Yaskawa INFORM job: DEMO_ROOF_SIDE_0625_3PAINT_60.JBI

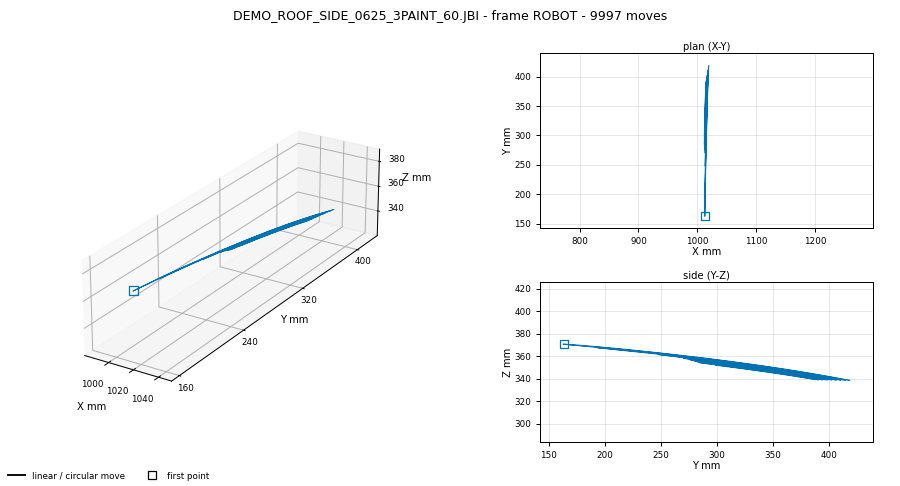
[picture p0: tool path of DEMO_ROOF_SIDE_0625_3PAINT_60.JBI in frame ROBOT, 9997 of 9997 moves have a stored position in this frame; points joined in program order, loops and branches not executed]
/JOB
//NAME DEMO_ROOF_SIDE_0625_3PAINT60
//POS
///NPOS 9997,0,0,0,0,0
///TOOL 0
///USER 0
///POSTYPE ROBOT
///RECTAN
///RCONF 1,0,0,0,0,0,0,0,0,0,0,0,0,0,0,0,0,0,0,0,0,0,0,0
C00000=1012.769,163.450,371.044,166.546,56.934,160.427
C00001=1012.773,163.699,371.026,166.549,56.922,160.426
C00002=1012.776,163.949,371.006,166.553,56.910,160.424
C00003=1012.781,164.198,370.986,166.556,56.898,160.423
C00004=1012.783,164.447,370.967,166.560,56.886,160.421
C00005=1012.788,164.696,370.948,166.563,56.875,160.420
C00006=1012.791,164.945,370.928,166.568,56.863,160.418
C00007=1012.795,165.195,370.908,166.571,56.851,160.417
C00008=1012.798,165.444,370.889,166.574,56.839,160.415
C00009=1012.802,165.693,370.869,166.578,56.827,160.414
C00010=1012.806,165.942,370.850,166.581,56.815,160.412
C00011=1012.810,166.191,370.830,166.586,56.803,160.411
C00012=1012.813,166.441,370.811,166.589,56.791,160.409
C00013=1012.817,166.690,370.791,166.592,56.779,160.408
C00014=1012.820,166.939,370.771,166.596,56.767,160.406
C00015=1012.825,167.188,370.752,166.599,56.756,160.405
C00016=1012.828,167.437,370.733,166.604,56.743,160.403
C00017=1012.832,167.686,370.713,166.607,56.732,160.402
C00018=1012.836,167.936,370.693,166.610,56.720,160.400
C00019=1012.839,168.185,370.673,166.614,56.707,160.398
C00020=1012.843,168.434,370.654,166.617,56.695,160.397
C00021=1012.846,168.684,370.635,166.621,56.683,160.395
C00022=1012.851,168.933,370.615,166.624,56.671,160.394
C00023=1012.854,169.182,370.595,166.629,56.659,160.393
C00024=1012.858,169.431,370.575,166.632,56.647,160.391
C00025=1012.862,169.680,370.556,166.636,56.635,160.390
C00026=1012.866,169.930,370.536,166.639,56.623,160.388
C00027=1012.870,170.208,370.514,166.644,56.609,160.386
C00028=1012.874,170.487,370.492,166.648,56.596,160.385
C00029=1012.878,170.766,370.470,166.652,56.583,160.383
C00030=1012.882,171.045,370.448,166.656,56.569,160.381
C00031=1012.887,171.294,370.428,166.661,56.557,160.380
C00032=1012.890,171.543,370.408,166.664,56.545,160.378
C00033=1012.894,171.793,370.389,166.668,56.532,160.377
C00034=1012.898,172.042,370.369,166.671,56.521,160.375
C00035=1012.902,172.292,370.349,166.675,56.509,160.374
C00036=1012.906,172.541,370.330,166.678,56.497,160.372
C00037=1012.910,172.790,370.310,166.683,56.485,160.371
C00038=1012.913,173.040,370.290,166.687,56.472,160.369
C00039=1012.917,173.288,370.271,166.690,56.460,160.367
C00040=1012.921,173.537,370.251,166.694,56.448,160.366
C00041=1012.925,173.786,370.231,166.699,56.436,160.365
C00042=1012.928,174.036,370.211,166.701,56.424,160.363
C00043=1012.932,174.285,370.191,166.706,56.411,160.361
C00044=1012.936,174.534,370.172,166.710,56.399,160.360
C00045=1012.940,174.783,370.151,166.713,56.388,160.358
C00046=1012.944,175.032,370.132,166.717,56.375,160.357
C00047=1012.948,175.282,370.112,166.721,56.363,160.355
C00048=1012.952,175.531,370.092,166.725,56.351,160.354
C00049=1012.956,175.780,370.072,166.729,56.339,160.352
C00050=1012.960,176.030,370.052,166.733,56.326,160.351
C00051=1012.964,176.279,370.033,166.737,56.314,160.349
C00052=1012.968,176.527,370.012,166.741,56.302,160.348
C00053=1012.972,176.776,369.993,166.744,56.289,160.346
C00054=1012.976,177.026,369.973,166.749,56.277,160.345
C00055=1012.979,177.275,369.952,166.753,56.265,160.343
C00056=1012.984,177.524,369.933,166.757,56.252,160.342
C00057=1012.987,177.773,369.913,166.760,56.241,160.340
C00058=1012.992,178.022,369.893,166.765,56.229,160.339
C00059=1012.995,178.272,369.873,166.769,56.216,160.337
C00060=1012.999,178.521,369.853,166.773,56.204,160.336
C00061=1013.004,178.770,369.833,166.777,56.191,160.334
C00062=1013.007,179.019,369.813,166.780,56.179,160.332
C00063=1013.012,179.268,369.794,166.785,56.167,160.331
C00064=1013.015,179.517,369.774,166.788,56.155,160.329
C00065=1013.019,179.767,369.753,166.793,56.142,160.328
C00066=1013.023,180.016,369.734,166.797,56.130,160.326
C00067=1013.028,180.265,369.713,166.801,56.118,160.325
C00068=1013.032,180.514,369.693,166.805,56.105,160.323
C00069=1013.036,180.764,369.673,166.809,56.093,160.322
C00070=1013.039,181.013,369.653,166.813,56.081,160.320
C00071=1013.044,181.261,369.633,166.817,56.068,160.319
C00072=1013.047,181.511,369.613,166.821,56.056,160.317
C00073=1013.050,181.760,369.592,166.826,56.044,160.316
C00074=1013.055,182.010,369.571,166.830,56.032,160.314
C00075=1013.059,182.259,369.550,166.833,56.020,160.313
C00076=1013.062,182.508,369.530,166.837,56.008,160.311
C00077=1013.066,182.757,369.509,166.842,55.996,160.310
C00078=1013.069,183.006,369.489,166.846,55.984,160.309
C00079=1013.073,183.255,369.468,166.849,55.972,160.307
C00080=1013.076,183.504,369.447,166.854,55.960,160.306
C00081=1013.080,183.753,369.427,166.858,55.947,160.304
C00082=1013.084,184.003,369.406,166.863,55.935,160.303
C00083=1013.088,184.252,369.385,166.866,55.924,160.301
C00084=1013.091,184.501,369.363,166.870,55.911,160.300
C00085=1013.095,184.750,369.343,166.874,55.899,160.298
C00086=1013.099,184.999,369.323,166.879,55.887,160.297
C00087=1013.103,185.247,369.302,166.883,55.874,160.295
C00088=1013.106,185.497,369.281,166.887,55.862,160.294
C00089=1013.110,185.747,369.260,166.891,55.851,160.292
C00090=1013.114,185.995,369.239,166.895,55.839,160.291
C00091=1013.118,186.274,369.216,166.900,55.825,160.289
C00092=1013.122,186.553,369.192,166.904,55.811,160.287
C00093=1013.127,186.832,369.169,166.910,55.798,160.286
C00094=1013.131,187.111,369.146,166.915,55.784,160.284
C00095=1013.134,187.360,369.125,166.918,55.772,160.283
C00096=1013.139,187.610,369.104,166.922,55.759,160.281
C00097=1013.142,187.858,369.083,166.927,55.748,160.280
C00098=1013.146,188.107,369.063,166.931,55.736,160.278
C00099=1013.150,188.356,369.041,166.935,55.723,160.277
C00100=1013.154,188.606,369.020,166.940,55.711,160.275
C00101=1013.158,188.854,368.999,166.944,55.699,160.274
C00102=1013.162,189.103,368.979,166.948,55.686,160.272
C00103=1013.165,189.353,368.958,166.953,55.674,160.271
C00104=1013.169,189.602,368.937,166.957,55.662,160.270
C00105=1013.173,189.851,368.916,166.961,55.650,160.268
C00106=1013.176,190.100,368.895,166.966,55.638,160.267
C00107=1013.181,190.349,368.874,166.970,55.625,160.265
C00108=1013.185,190.598,368.853,166.975,55.613,160.264
C00109=1013.189,190.847,368.832,166.979,55.601,160.262
C00110=1013.192,191.097,368.810,166.983,55.588,160.261
C00111=1013.196,191.345,368.789,166.988,55.576,160.259
C00112=1013.200,191.594,368.769,166.992,55.564,160.258
C00113=1013.205,191.843,368.747,166.996,55.552,160.256
C00114=1013.208,192.092,368.726,167.001,55.540,160.255
C00115=1013.212,192.341,368.705,167.005,55.527,160.253
C00116=1013.216,192.591,368.684,167.010,55.515,160.252
C00117=1013.220,192.840,368.663,167.015,55.502,160.251
C00118=1013.224,193.088,368.642,167.019,55.490,160.249
C00119=1013.228,193.338,368.621,167.023,55.478,160.248
C00120=1013.232,193.587,368.600,167.028,55.466,160.246
C00121=1013.236,193.836,368.578,167.033,55.454,160.245
C00122=1013.240,194.085,368.558,167.037,55.441,160.243
C00123=1013.244,194.334,368.537,167.041,55.429,160.242
C00124=1013.248,194.583,368.516,167.045,55.417,160.240
C00125=1013.251,194.832,368.494,167.051,55.404,160.239
C00126=1013.256,195.082,368.473,167.055,55.392,160.237
C00127=1013.260,195.330,368.452,167.060,55.380,160.236
C00128=1013.263,195.580,368.431,167.064,55.367,160.234
C00129=1013.267,195.829,368.410,167.068,55.355,160.233
C00130=1013.271,196.078,368.389,167.073,55.343,160.231
C00131=1013.276,196.326,368.367,167.078,55.331,160.230
C00132=1013.279,196.576,368.346,167.082,55.318,160.229
C00133=1013.284,196.825,368.325,167.087,55.306,160.227
C00134=1013.288,197.074,368.304,167.091,55.293,160.226
C00135=1013.292,197.323,368.283,167.097,55.281,160.224
C00136=1013.295,197.572,368.261,167.101,55.269,160.223
C00137=1013.300,197.821,368.239,167.106,55.257,160.221
C00138=1013.304,198.070,368.219,167.110,55.244,160.220
C00139=1013.308,198.319,368.197,167.115,55.232,160.219
C00140=1013.312,198.568,368.176,167.120,55.219,160.217
C00141=1013.316,198.818,368.155,167.124,55.207,160.216
C00142=1013.320,199.067,368.133,167.128,55.195,160.214
C00143=1013.324,199.316,368.111,167.134,55.183,160.213
C00144=1013.328,199.565,368.089,167.138,55.170,160.211
C00145=1013.332,199.814,368.068,167.143,55.158,160.210
C00146=1013.336,200.063,368.045,167.148,55.146,160.209
C00147=1013.340,200.312,368.025,167.152,55.134,160.207
C00148=1013.344,200.561,368.002,167.157,55.122,160.206
C00149=1013.347,200.810,367.981,167.162,55.109,160.204
C00150=1013.352,201.059,367.959,167.166,55.097,160.203
C00151=1013.356,201.308,367.937,167.171,55.085,160.201
C00152=1013.359,201.557,367.915,167.176,55.072,160.200
C00153=1013.364,201.806,367.894,167.181,55.061,160.199
C00154=1013.367,202.055,367.872,167.185,55.048,160.197
C00155=1013.384,203.102,367.780,167.720,55.151,160.345
C00156=1013.390,203.386,367.754,167.725,55.138,160.343
C00157=1013.395,203.671,367.727,167.730,55.125,160.342
C00158=1013.402,203.957,367.700,167.736,55.113,160.340
C00159=1013.408,204.241,367.672,167.741,55.100,160.339
C00160=1013.412,204.490,367.649,167.746,55.089,160.337
C00161=1013.417,204.739,367.626,167.751,55.077,160.336
C00162=1013.422,204.988,367.602,167.755,55.066,160.335
C00163=1013.428,205.237,367.579,167.760,55.055,160.333
C00164=1013.433,205.486,367.555,167.764,55.045,160.332
C00165=1013.438,205.734,367.531,167.769,55.034,160.331
C00166=1013.443,205.983,367.508,167.773,55.022,160.329
C00167=1013.448,206.232,367.484,167.778,55.011,160.328
C00168=1013.453,206.481,367.460,167.782,55.001,160.327
C00169=1013.458,206.730,367.436,167.787,54.989,160.326
C00170=1013.463,206.978,367.412,167.791,54.979,160.324
C00171=1013.468,207.227,367.389,167.796,54.968,160.323
C00172=1013.473,207.476,367.365,167.800,54.957,160.322
C00173=1013.478,207.725,367.341,167.806,54.946,160.320
C00174=1013.483,207.973,367.317,167.810,54.935,160.319
C00175=1013.488,208.223,367.293,167.815,54.924,160.318
C00176=1013.493,208.451,367.271,167.818,54.914,160.316
C00177=1013.498,208.678,367.250,167.822,54.904,160.315
C00178=1013.502,208.907,367.228,167.827,54.894,160.314
C00179=1013.507,209.134,367.206,167.831,54.885,160.313
C00180=1013.511,209.362,367.184,167.835,54.875,160.312
C00181=1013.516,209.590,367.161,167.840,54.865,160.311
C00182=1013.520,209.818,367.139,167.844,54.855,160.310
C00183=1013.525,210.046,367.118,167.848,54.845,160.309
C00184=1013.530,210.294,367.093,167.852,54.835,160.307
C00185=1013.535,210.544,367.069,167.856,54.824,160.306
C00186=1013.540,210.792,367.045,167.862,54.813,160.305
C00187=1013.545,211.041,367.021,167.866,54.802,160.303
C00188=1013.550,211.290,366.997,167.871,54.791,160.302
C00189=1013.555,211.539,366.972,167.875,54.781,160.301
C00190=1013.560,211.788,366.948,167.880,54.771,160.300
C00191=1013.565,212.036,366.924,167.885,54.760,160.299
C00192=1013.570,212.285,366.900,167.889,54.749,160.297
C00193=1013.576,212.534,366.876,167.893,54.739,160.296
C00194=1013.580,212.783,366.851,167.898,54.728,160.295
C00195=1013.586,213.032,366.827,167.903,54.718,160.294
C00196=1013.591,213.280,366.803,167.907,54.707,160.292
C00197=1013.596,213.529,366.779,167.911,54.697,160.291
C00198=1013.601,213.778,366.755,167.917,54.686,160.290
C00199=1013.606,214.027,366.730,167.921,54.676,160.289
C00200=1013.611,214.275,366.706,167.925,54.665,160.287
C00201=1013.616,214.524,366.681,167.931,54.654,160.286
C00202=1013.622,214.773,366.657,167.935,54.644,160.285
C00203=1013.626,215.021,366.632,167.939,54.634,160.284
C00204=1013.631,215.271,366.609,167.944,54.623,160.282
C00205=1013.636,215.519,366.585,167.949,54.613,160.281
C00206=1013.642,215.769,366.560,167.954,54.602,160.280
C00207=1013.648,216.017,366.536,167.958,54.592,160.279
C00208=1013.652,216.266,366.511,167.963,54.581,160.278
C00209=1013.657,216.515,366.487,167.968,54.571,160.277
C00210=1013.663,216.763,366.462,167.972,54.561,160.275
C00211=1013.668,217.012,366.438,167.977,54.550,160.274
C00212=1013.673,217.261,366.413,167.982,54.539,160.273
C00213=1013.678,217.509,366.389,167.987,54.529,160.272
C00214=1013.683,217.758,366.365,167.991,54.519,160.271
C00215=1013.688,218.007,366.340,167.995,54.509,160.269
C00216=1013.694,218.258,366.315,168.000,54.498,160.268
C00217=1013.699,218.511,366.289,168.005,54.488,160.267
C00218=1013.704,218.764,366.264,168.010,54.478,160.266
C00219=1013.709,219.015,366.239,168.014,54.468,160.265
C00220=1013.714,219.263,366.215,168.019,54.457,160.263
C00221=1013.719,219.513,366.189,168.023,54.447,160.262
C00222=1013.724,219.762,366.165,168.028,54.437,160.261
C00223=1013.729,220.010,366.140,168.033,54.427,160.260
C00224=1013.735,220.259,366.115,168.038,54.417,160.259
C00225=1013.739,220.507,366.090,168.043,54.407,160.258
C00226=1013.745,220.757,366.066,168.047,54.396,160.257
C00227=1013.750,221.005,366.040,168.052,54.386,160.256
C00228=1013.755,221.254,366.016,168.056,54.377,160.254
C00229=1013.760,221.503,365.991,168.061,54.367,160.253
C00230=1013.765,221.750,365.966,168.065,54.356,160.252
C00231=1013.770,222.000,365.941,168.070,54.346,160.251
C00232=1013.776,222.249,365.917,168.075,54.337,160.250
C00233=1013.781,222.497,365.891,168.080,54.327,160.249
C00234=1013.786,222.746,365.867,168.084,54.316,160.247
C00235=1013.791,222.995,365.842,168.090,54.306,160.247
C00236=1013.797,223.243,365.817,168.094,54.296,160.245
C00237=1013.801,223.492,365.792,168.099,54.286,160.244
C00238=1013.807,223.741,365.767,168.104,54.277,160.243
C00239=1013.812,223.990,365.742,168.108,54.266,160.242
C00240=1013.817,224.238,365.717,168.113,54.256,160.241
C00241=1013.823,224.487,365.692,168.118,54.246,160.240
C00242=1013.827,224.736,365.667,168.122,54.237,160.239
C00243=1013.833,224.984,365.642,168.127,54.227,160.238
C00244=1013.838,225.234,365.616,168.132,54.217,160.237
C00245=1013.844,225.482,365.592,168.137,54.207,160.236
C00246=1013.848,225.730,365.567,168.141,54.197,160.234
C00247=1013.854,225.979,365.541,168.146,54.187,160.233
C00248=1013.859,226.228,365.516,168.151,54.177,160.232
C00249=1013.864,226.476,365.491,168.156,54.168,160.231
C00250=1013.869,226.725,365.465,168.161,54.158,160.230
C00251=1013.875,226.974,365.441,168.165,54.148,160.229
C00252=1013.880,227.223,365.415,168.170,54.139,160.228
C00253=1013.885,227.471,365.389,168.174,54.129,160.227
C00254=1013.890,227.720,365.364,168.179,54.119,160.226
C00255=1013.895,227.969,365.338,168.184,54.110,160.225
C00256=1013.901,228.217,365.313,168.188,54.100,160.224
C00257=1013.906,228.466,365.288,168.193,54.090,160.222
C00258=1013.911,228.715,365.263,168.198,54.080,160.221
C00259=1013.916,228.963,365.237,168.203,54.071,160.221
C00260=1013.922,229.212,365.212,168.208,54.061,160.219
C00261=1013.927,229.460,365.186,168.213,54.052,160.218
C00262=1013.932,229.709,365.160,168.217,54.042,160.217
C00263=1013.937,229.957,365.135,168.222,54.033,160.216
C00264=1013.942,230.206,365.110,168.227,54.023,160.215
C00265=1013.947,230.455,365.084,168.231,54.014,160.214
C00266=1013.952,230.704,365.058,168.236,54.004,160.213
C00267=1013.957,230.952,365.032,168.242,53.995,160.212
C00268=1013.962,231.201,365.007,168.245,53.985,160.211
C00269=1013.968,231.450,364.981,168.250,53.976,160.210
C00270=1013.973,231.698,364.955,168.256,53.967,160.209
C00271=1013.978,231.947,364.929,168.260,53.957,160.208
C00272=1013.983,232.195,364.904,168.265,53.947,160.207
C00273=1013.989,232.444,364.879,168.269,53.938,160.206
C00274=1013.994,232.692,364.853,168.274,53.929,160.205
C00275=1013.999,232.941,364.827,168.280,53.920,160.204
C00276=1014.005,233.188,364.802,168.284,53.910,160.203
C00277=1014.010,233.433,364.776,168.289,53.901,160.202
C00278=1014.014,233.680,364.750,168.294,53.892,160.201
C00279=1014.020,233.927,364.725,168.299,53.882,160.200
C00280=1014.025,234.173,364.699,168.303,53.873,160.199
C00281=1014.030,234.419,364.674,168.308,53.864,160.198
C00282=1014.036,234.665,364.648,168.313,53.854,160.197
C00283=1014.041,234.911,364.622,168.317,53.846,160.196
C00284=1014.046,235.159,364.597,168.322,53.836,160.195
C00285=1014.051,235.408,364.571,168.327,53.827,160.194
C00286=1014.057,235.657,364.544,168.333,53.818,160.193
C00287=1014.062,235.905,364.519,168.336,53.809,160.192
C00288=1014.067,236.154,364.493,168.342,53.800,160.191
C00289=1014.073,236.403,364.467,168.347,53.790,160.190
C00290=1014.078,236.651,364.441,168.351,53.781,160.189
C00291=1014.083,236.900,364.415,168.356,53.772,160.189
C00292=1014.089,237.149,364.389,168.361,53.762,160.187
C00293=1014.094,237.397,364.363,168.365,53.754,160.186
C00294=1014.099,237.646,364.337,168.370,53.744,160.185
C00295=1014.105,237.894,364.311,168.376,53.735,160.185
C00296=1014.110,238.143,364.285,168.381,53.726,160.184
C00297=1014.115,238.392,364.259,168.385,53.717,160.183
C00298=1014.121,238.639,364.233,168.390,53.708,160.182
C00299=1014.126,238.888,364.207,168.395,53.699,160.181
C00300=1014.131,239.137,364.180,168.400,53.690,160.180
C00301=1014.136,239.386,364.154,168.405,53.681,160.179
C00302=1014.142,239.633,364.127,168.410,53.673,160.178
C00303=1014.146,239.883,364.101,168.414,53.663,160.177
C00304=1014.152,240.131,364.074,168.419,53.654,160.176
C00305=1014.157,240.379,364.049,168.424,53.645,160.175
C00306=1014.163,240.628,364.022,168.430,53.636,160.174
C00307=1014.168,240.877,363.995,168.434,53.628,160.173
C00308=1014.173,241.125,363.969,168.439,53.619,160.173
C00309=1014.178,241.374,363.943,168.444,53.610,160.172
C00310=1014.183,241.622,363.916,168.449,53.601,160.171
C00311=1014.189,241.871,363.889,168.453,53.592,160.170
C00312=1014.194,242.120,363.863,168.459,53.583,160.169
C00313=1014.200,242.367,363.837,168.464,53.574,160.168
C00314=1014.205,242.616,363.810,168.468,53.566,160.167
C00315=1014.210,242.865,363.784,168.474,53.557,160.166
C00316=1014.215,243.114,363.757,168.478,53.548,160.165
C00317=1014.221,243.362,363.730,168.482,53.540,160.164
C00318=1014.225,243.610,363.703,168.488,53.531,160.164
C00319=1014.231,243.858,363.677,168.493,53.523,160.163
C00320=1014.236,244.107,363.649,168.498,53.514,160.162
C00321=1014.241,244.356,363.623,168.502,53.505,160.161
C00322=1014.247,244.605,363.596,168.508,53.496,160.160
C00323=1014.252,244.853,363.569,168.512,53.488,160.159
C00324=1014.257,245.101,363.543,168.518,53.479,160.159
C00325=1014.262,245.350,363.515,168.522,53.471,160.158
C00326=1014.267,245.598,363.488,168.527,53.462,160.157
C00327=1014.273,245.847,363.461,168.532,53.453,160.156
C00328=1014.278,246.095,363.434,168.537,53.445,160.155
C00329=1014.284,246.344,363.408,168.542,53.436,160.154
C00330=1014.289,246.592,363.380,168.547,53.428,160.153
C00331=1014.294,246.841,363.353,168.553,53.420,160.153
C00332=1014.299,247.089,363.326,168.557,53.411,160.152
C00333=1014.304,247.337,363.300,168.561,53.403,160.151
C00334=1014.310,247.586,363.273,168.567,53.394,160.150
C00335=1014.315,247.834,363.246,168.572,53.386,160.149
C00336=1014.320,248.077,363.220,168.577,53.378,160.149
C00337=1014.325,248.321,363.193,168.582,53.369,160.148
C00338=1014.331,248.563,363.167,168.587,53.361,160.147
C00339=1014.336,248.806,363.140,168.591,53.352,160.146
C00340=1014.341,249.049,363.115,168.596,53.345,160.145
C00341=1014.346,249.291,363.087,168.600,53.336,160.144
C00342=1014.352,249.534,363.061,168.606,53.328,160.144
C00343=1014.356,249.777,363.035,168.611,53.320,160.143
C00344=1014.362,250.025,363.008,168.616,53.311,160.142
C00345=1014.367,250.274,362.981,168.621,53.303,160.142
C00346=1014.373,250.522,362.953,168.626,53.295,160.141
C00347=1014.378,250.770,362.926,168.631,53.287,160.140
C00348=1014.383,251.019,362.899,168.636,53.278,160.139
C00349=1014.389,251.267,362.872,168.641,53.270,160.138
C00350=1014.394,251.516,362.845,168.645,53.261,160.137
C00351=1014.400,251.765,362.817,168.651,53.253,160.137
C00352=1014.406,252.013,362.790,168.656,53.245,160.136
C00353=1014.411,252.262,362.763,168.662,53.236,160.135
C00354=1014.417,252.510,362.736,168.667,53.229,160.134
C00355=1014.422,252.759,362.709,168.671,53.220,160.134
C00356=1014.427,253.007,362.681,168.677,53.212,160.133
C00357=1014.433,253.255,362.654,168.681,53.203,160.132
C00358=1014.438,253.504,362.627,168.686,53.195,160.131
C00359=1014.444,253.752,362.600,168.692,53.187,160.131
C00360=1014.450,254.001,362.572,168.696,53.179,160.130
C00361=1014.455,254.250,362.545,168.701,53.171,160.129
C00362=1014.461,254.497,362.517,168.707,53.163,160.128
C00363=1014.466,254.746,362.490,168.712,53.155,160.128
C00364=1014.472,254.994,362.464,168.717,53.146,160.127
C00365=1014.477,255.243,362.436,168.722,53.138,160.126
C00366=1014.483,255.492,362.408,168.727,53.130,160.125
C00367=1014.489,255.740,362.381,168.732,53.122,160.124
C00368=1014.494,255.988,362.353,168.738,53.114,160.124
C00369=1014.499,256.237,362.327,168.743,53.106,160.123
C00370=1014.505,256.485,362.298,168.747,53.098,160.122
C00371=1014.510,256.734,362.271,168.753,53.090,160.122
C00372=1014.516,256.982,362.244,168.758,53.081,160.121
C00373=1014.522,257.231,362.217,168.763,53.073,160.120
C00374=1014.527,257.479,362.188,168.768,53.066,160.119
C00375=1014.533,257.728,362.162,168.773,53.057,160.119
C00376=1014.539,257.976,362.134,168.778,53.050,160.118
C00377=1014.545,258.225,362.107,168.783,53.042,160.117
C00378=1014.550,258.473,362.079,168.789,53.034,160.117
C00379=1014.555,258.721,362.051,168.794,53.026,160.116
C00380=1014.561,258.969,362.024,168.799,53.017,160.115
C00381=1014.567,259.218,361.996,168.803,53.009,160.114
C00382=1014.573,259.466,361.968,168.809,53.001,160.114
C00383=1014.578,259.714,361.941,168.814,52.993,160.113
C00384=1014.584,259.962,361.913,168.820,52.986,160.112
C00385=1014.590,260.211,361.885,168.825,52.979,160.112
C00386=1014.595,260.459,361.857,168.829,52.971,160.111
C00387=1014.600,260.707,361.829,168.835,52.963,160.110
C00388=1014.606,260.956,361.801,168.840,52.955,160.110
C00389=1014.611,261.205,361.773,168.845,52.947,160.109
C00390=1014.617,261.453,361.745,168.851,52.940,160.108
C00391=1014.623,261.701,361.717,168.856,52.932,160.108
C00392=1014.627,261.950,361.689,168.860,52.924,160.107
C00393=1014.633,262.198,361.661,168.865,52.916,160.106
C00394=1014.639,262.447,361.632,168.872,52.909,160.106
C00395=1014.644,262.695,361.604,168.877,52.901,160.105
C00396=1014.650,262.936,361.577,168.882,52.893,160.104
C00397=1014.655,263.178,361.550,168.887,52.886,160.104
C00398=1014.660,263.420,361.522,168.892,52.879,160.103
C00399=1014.666,263.662,361.495,168.896,52.872,160.102
C00400=1014.671,263.903,361.467,168.901,52.864,160.102
C00401=1014.677,264.146,361.440,168.907,52.857,160.101
C00402=1014.682,264.387,361.413,168.912,52.849,160.100
C00403=1014.687,264.629,361.385,168.917,52.842,160.100
C00404=1014.693,264.877,361.356,168.922,52.834,160.099
C00405=1014.699,265.125,361.328,168.927,52.827,160.099
C00406=1014.705,265.374,361.300,168.932,52.819,160.098
C00407=1014.710,265.622,361.272,168.938,52.812,160.097
C00408=1014.716,265.871,361.243,168.944,52.804,160.097
C00409=1014.721,266.119,361.215,168.949,52.797,160.096
C00410=1014.727,266.367,361.186,168.954,52.789,160.096
C00411=1014.732,266.615,361.158,168.959,52.782,160.095
C00412=1014.738,266.864,361.129,168.964,52.774,160.094
C00413=1014.744,267.112,361.101,168.970,52.767,160.094
C00414=1014.749,267.361,361.072,168.975,52.760,160.093
C00415=1014.755,267.608,361.044,168.980,52.753,160.093
C00416=1014.761,267.857,361.015,168.985,52.745,160.092
C00417=1014.767,268.106,360.987,168.990,52.738,160.091
C00418=1014.771,268.353,360.958,168.996,52.731,160.091
C00419=1014.777,268.602,360.929,169.001,52.724,160.090
C00420=1014.783,268.850,360.901,169.006,52.716,160.090
C00421=1014.789,269.098,360.872,169.011,52.709,160.089
C00422=1014.794,269.347,360.844,169.017,52.702,160.089
C00423=1014.800,269.595,360.815,169.022,52.695,160.088
C00424=1014.806,269.844,360.787,169.027,52.687,160.087
C00425=1014.811,270.091,360.757,169.033,52.680,160.087
C00426=1014.817,270.340,360.729,169.038,52.673,160.086
C00427=1014.822,270.588,360.699,169.043,52.666,160.086
C00428=1014.827,270.837,360.671,169.049,52.659,160.085
C00429=1014.834,271.085,360.642,169.054,52.652,160.085
C00430=1014.839,271.332,360.613,169.059,52.644,160.084
C00431=1014.845,271.581,360.585,169.065,52.637,160.084
C00432=1014.851,271.829,360.556,169.070,52.630,160.083
C00433=1014.856,272.077,360.526,169.075,52.623,160.083
C00434=1014.862,272.326,360.498,169.081,52.616,160.082
C00435=1014.867,272.574,360.468,169.086,52.608,160.082
C00436=1014.873,272.822,360.439,169.092,52.601,160.081
C00437=1014.878,273.071,360.411,169.097,52.594,160.081
C00438=1014.884,273.319,360.382,169.102,52.587,160.080
C00439=1014.890,273.567,360.352,169.108,52.580,160.080
C00440=1014.895,273.815,360.323,169.113,52.573,160.079
C00441=1014.901,274.064,360.295,169.119,52.566,160.079
C00442=1014.907,274.312,360.266,169.124,52.559,160.078
C00443=1014.913,274.560,360.236,169.129,52.552,160.078
C00444=1014.918,274.808,360.207,169.135,52.545,160.077
C00445=1014.924,275.056,360.178,169.140,52.538,160.077
C00446=1014.930,275.304,360.149,169.146,52.531,160.076
C00447=1014.936,275.553,360.120,169.151,52.524,160.076
C00448=1014.941,275.802,360.091,169.157,52.517,160.075
C00449=1014.947,276.049,360.062,169.162,52.511,160.075
C00450=1014.952,276.297,360.032,169.168,52.504,160.074
C00451=1014.958,276.546,360.003,169.172,52.497,160.074
C00452=1014.964,276.794,359.974,169.178,52.490,160.073
C00453=1014.970,277.042,359.943,169.184,52.483,160.073
C00454=1014.975,277.290,359.914,169.189,52.476,160.072
C00455=1014.980,277.538,359.884,169.194,52.469,160.072
C00456=1014.986,277.782,359.856,169.200,52.463,160.072
C00457=1014.992,278.027,359.827,169.205,52.456,160.071
C00458=1014.998,278.270,359.798,169.211,52.450,160.071
C00459=1015.003,278.514,359.769,169.216,52.443,160.070
C00460=1015.009,278.758,359.739,169.222,52.437,160.070
C00461=1015.014,279.002,359.710,169.226,52.430,160.069
C00462=1015.020,279.247,359.682,169.232,52.424,160.069
C00463=1015.026,279.490,359.652,169.238,52.417,160.068
C00464=1015.031,279.739,359.622,169.243,52.410,160.068
C00465=1015.038,279.987,359.593,169.249,52.403,160.068
C00466=1015.043,280.235,359.563,169.254,52.396,160.067
C00467=1015.049,280.483,359.533,169.259,52.390,160.067
C00468=1015.054,280.732,359.504,169.265,52.383,160.066
C00469=1015.061,280.980,359.475,169.270,52.377,160.066
C00470=1015.067,281.228,359.444,169.276,52.370,160.065
C00471=1015.072,281.476,359.415,169.282,52.364,160.065
C00472=1015.077,281.724,359.386,169.287,52.357,160.065
C00473=1015.084,281.972,359.355,169.293,52.350,160.064
C00474=1015.090,282.220,359.326,169.298,52.344,160.064
C00475=1015.095,282.469,359.296,169.303,52.337,160.063
C00476=1015.102,282.716,359.266,169.309,52.331,160.063
C00477=1015.107,282.965,359.237,169.315,52.324,160.063
C00478=1015.113,283.213,359.206,169.321,52.318,160.062
C00479=1015.119,283.461,359.177,169.326,52.311,160.062
C00480=1015.125,283.709,359.147,169.332,52.304,160.061
C00481=1015.131,283.957,359.117,169.337,52.298,160.061
C00482=1015.136,284.205,359.087,169.343,52.292,160.061
C00483=1015.142,284.453,359.057,169.348,52.285,160.060
C00484=1015.148,284.701,359.027,169.354,52.279,160.060
C00485=1015.154,284.949,358.997,169.360,52.272,160.060
C00486=1015.159,285.197,358.967,169.366,52.266,160.059
C00487=1015.166,285.445,358.937,169.370,52.259,160.059
C00488=1015.171,285.693,358.907,169.376,52.253,160.058
C00489=1015.178,285.942,358.877,169.382,52.247,160.058
C00490=1015.183,286.190,358.847,169.388,52.240,160.058
C00491=1015.189,286.438,358.816,169.394,52.234,160.058
C00492=1015.195,286.686,358.787,169.399,52.228,160.057
C00493=1015.201,286.934,358.756,169.405,52.222,160.057
C00494=1015.206,287.182,358.726,169.410,52.216,160.057
C00495=1015.212,287.429,358.696,169.416,52.209,160.056
C00496=1015.219,287.678,358.665,169.422,52.203,160.056
C00497=1015.224,287.926,358.634,169.427,52.197,160.056
C00498=1015.230,288.174,358.605,169.433,52.191,160.055
C00499=1015.236,288.422,358.575,169.439,52.184,160.055
C00500=1015.242,288.670,358.544,169.445,52.178,160.055
C00501=1015.248,288.918,358.513,169.450,52.172,160.054
C00502=1015.254,289.166,358.483,169.456,52.166,160.054
C00503=1015.259,289.414,358.452,169.461,52.160,160.054
C00504=1015.265,289.662,358.422,169.467,52.153,160.053
C00505=1015.271,289.911,358.391,169.472,52.147,160.053
C00506=1015.277,290.159,358.361,169.478,52.141,160.053
C00507=1015.283,290.406,358.330,169.484,52.135,160.052
C00508=1015.289,290.655,358.300,169.490,52.128,160.052
C00509=1015.295,290.903,358.269,169.496,52.123,160.052
C00510=1015.301,291.151,358.239,169.501,52.117,160.052
C00511=1015.307,291.398,358.209,169.507,52.111,160.051
C00512=1015.313,291.647,358.178,169.513,52.104,160.051
C00513=1015.318,291.894,358.146,169.519,52.099,160.051
C00514=1015.324,292.142,358.116,169.524,52.093,160.050
C00515=1015.331,292.391,358.085,169.530,52.086,160.050
C00516=1015.336,292.643,358.054,169.536,52.080,160.050
C00517=1015.342,292.895,358.022,169.542,52.075,160.050
C00518=1015.348,293.148,357.991,169.548,52.068,160.049
C00519=1015.355,293.400,357.959,169.553,52.063,160.049
C00520=1015.360,293.648,357.928,169.559,52.057,160.049
C00521=1015.366,293.896,357.897,169.566,52.051,160.049
C00522=1015.371,294.144,357.866,169.571,52.045,160.049
C00523=1015.378,294.392,357.835,169.577,52.040,160.048
C00524=1015.383,294.640,357.804,169.583,52.033,160.048
C00525=1015.389,294.888,357.772,169.588,52.028,160.048
C00526=1015.394,295.136,357.742,169.594,52.022,160.048
C00527=1015.401,295.384,357.710,169.600,52.016,160.048
C00528=1015.407,295.631,357.678,169.606,52.011,160.047
C00529=1015.412,295.879,357.648,169.612,52.005,160.047
C00530=1015.418,296.127,357.616,169.618,51.999,160.047
C00531=1015.424,296.375,357.586,169.623,51.993,160.047
C00532=1015.430,296.623,357.554,169.629,51.987,160.046
C00533=1015.436,296.870,357.523,169.636,51.982,160.046
C00534=1015.442,297.119,357.491,169.640,51.976,160.046
C00535=1015.448,297.366,357.460,169.647,51.970,160.046
C00536=1015.454,297.615,357.428,169.653,51.965,160.046
C00537=1015.459,297.863,357.397,169.658,51.960,160.046
C00538=1015.466,298.111,357.366,169.664,51.953,160.045
C00539=1015.471,298.358,357.334,169.671,51.948,160.045
C00540=1015.478,298.606,357.303,169.676,51.942,160.045
C00541=1015.484,298.855,357.271,169.682,51.937,160.045
C00542=1015.490,299.102,357.240,169.688,51.931,160.045
C00543=1015.496,299.350,357.208,169.694,51.925,160.044
C00544=1015.502,299.598,357.177,169.700,51.920,160.044
C00545=1015.508,299.846,357.146,169.706,51.914,160.044
C00546=1015.514,300.094,357.115,169.712,51.909,160.044
C00547=1015.520,300.342,357.083,169.718,51.903,160.044
C00548=1015.526,300.590,357.051,169.724,51.898,160.044
C00549=1015.532,300.837,357.020,169.729,51.892,160.044
C00550=1015.539,301.085,356.988,169.736,51.886,160.043
C00551=1015.544,301.333,356.956,169.742,51.881,160.043
C00552=1015.550,301.581,356.925,169.747,51.875,160.043
C00553=1015.557,301.829,356.893,169.754,51.870,160.043
C00554=1015.563,302.077,356.861,169.760,51.864,160.043
C00555=1015.569,302.325,356.830,169.765,51.859,160.043
C00556=1015.575,302.572,356.798,169.772,51.853,160.043
C00557=1015.581,302.820,356.767,169.778,51.848,160.043
C00558=1015.587,303.069,356.735,169.783,51.843,160.042
C00559=1015.594,303.316,356.703,169.790,51.837,160.042
C00560=1015.600,303.564,356.672,169.796,51.831,160.042
C00561=1015.606,303.812,356.640,169.802,51.826,160.042
C00562=1015.612,304.060,356.608,169.808,51.821,160.042
C00563=1015.619,304.308,356.577,169.814,51.816,160.042
C00564=1015.624,304.555,356.545,169.821,51.810,160.042
C00565=1015.630,304.804,356.513,169.826,51.805,160.042
C00566=1015.637,305.051,356.481,169.832,51.799,160.042
C00567=1015.643,305.299,356.449,169.839,51.794,160.042
C00568=1015.650,305.547,356.417,169.844,51.789,160.041
C00569=1015.656,305.795,356.385,169.851,51.784,160.042
C00570=1015.663,306.043,356.354,169.857,51.778,160.041
C00571=1015.668,306.290,356.322,169.863,51.773,160.041
C00572=1015.675,306.538,356.290,169.869,51.767,160.041
C00573=1015.681,306.786,356.258,169.876,51.762,160.041
C00574=1015.688,307.033,356.226,169.882,51.757,160.041
C00575=1015.694,307.282,356.194,169.887,51.752,160.041
C00576=1015.701,307.552,356.159,169.895,51.746,160.041
C00577=1015.708,307.823,356.124,169.901,51.740,160.041
C00578=1015.715,308.092,356.089,169.907,51.735,160.041
C00579=1015.722,308.363,356.054,169.915,51.729,160.041
C00580=1015.729,308.610,356.022,169.922,51.724,160.041
C00581=1015.735,308.858,355.990,169.927,51.719,160.041
C00582=1015.741,309.106,355.959,169.933,51.713,160.041
C00583=1015.748,309.354,355.926,169.940,51.708,160.041
C00584=1015.754,309.601,355.893,169.945,51.703,160.040
C00585=1015.760,309.849,355.861,169.952,51.698,160.041
C00586=1015.766,310.097,355.828,169.958,51.693,160.041
C00587=1015.772,310.345,355.795,169.964,51.688,160.040
C00588=1015.778,310.593,355.762,169.970,51.683,160.041
C00589=1015.784,310.840,355.730,169.977,51.678,160.041
C00590=1015.791,311.088,355.697,169.984,51.674,160.041
C00591=1015.797,311.335,355.664,169.989,51.668,160.041
C00592=1015.803,311.583,355.631,169.996,51.663,160.041
C00593=1015.809,311.831,355.599,170.001,51.659,160.041
C00594=1015.815,312.079,355.566,170.008,51.654,160.041
C00595=1015.821,312.327,355.533,170.015,51.648,160.041
C00596=1015.827,312.574,355.501,170.020,51.644,160.041
C00597=1015.834,312.822,355.468,170.027,51.639,160.041
C00598=1015.839,313.070,355.434,170.033,51.635,160.041
C00599=1015.846,313.317,355.402,170.040,51.630,160.041
C00600=1015.852,313.566,355.369,170.046,51.625,160.041
C00601=1015.859,313.813,355.335,170.052,51.620,160.041
C00602=1015.865,314.060,355.302,170.059,51.615,160.041
C00603=1015.871,314.308,355.269,170.065,51.611,160.041
C00604=1015.877,314.556,355.236,170.072,51.606,160.041
C00605=1015.884,314.803,355.204,170.078,51.600,160.041
C00606=1015.890,315.052,355.170,170.084,51.596,160.041
C00607=1015.897,315.299,355.138,170.090,51.591,160.041
C00608=1015.902,315.547,355.104,170.096,51.586,160.041
C00609=1015.909,315.794,355.071,170.103,51.582,160.042
C00610=1015.915,316.042,355.038,170.110,51.577,160.042
C00611=1015.922,316.290,355.005,170.116,51.573,160.042
C00612=1015.928,316.537,354.972,170.123,51.568,160.042
C00613=1015.934,316.785,354.938,170.129,51.563,160.042
C00614=1015.940,317.032,354.906,170.135,51.558,160.042
C00615=1015.947,317.281,354.872,170.142,51.554,160.042
C00616=1015.954,317.528,354.839,170.148,51.549,160.042
C00617=1015.960,317.775,354.806,170.155,51.544,160.042
C00618=1015.966,318.024,354.773,170.161,51.539,160.042
C00619=1015.973,318.271,354.739,170.168,51.535,160.043
C00620=1015.979,318.518,354.706,170.174,51.531,160.043
C00621=1015.986,318.767,354.673,170.181,51.526,160.043
C00622=1015.993,319.014,354.640,170.187,51.521,160.043
C00623=1015.999,319.262,354.606,170.194,51.517,160.043
C00624=1016.006,319.509,354.573,170.200,51.512,160.043
C00625=1016.012,319.758,354.540,170.207,51.508,160.043
C00626=1016.019,320.004,354.506,170.213,51.503,160.043
C00627=1016.025,320.252,354.473,170.220,51.499,160.044
C00628=1016.032,320.500,354.439,170.226,51.494,160.044
C00629=1016.038,320.748,354.406,170.233,51.489,160.044
C00630=1016.045,320.995,354.372,170.239,51.485,160.044
C00631=1016.052,321.242,354.339,170.246,51.480,160.044
C00632=1016.058,321.491,354.305,170.253,51.476,160.045
C00633=1016.065,321.738,354.272,170.259,51.472,160.045
C00634=1016.072,321.986,354.239,170.266,51.467,160.045
C00635=1016.079,322.234,354.205,170.273,51.463,160.045
C00636=1016.086,322.509,354.167,170.280,51.458,160.045
C00637=1016.093,322.785,354.130,170.288,51.452,160.045
C00638=1016.100,323.061,354.092,170.294,51.448,160.045
C00639=1016.108,323.336,354.056,170.303,51.443,160.046
C00640=1016.115,323.584,354.021,170.309,51.438,160.046
C00641=1016.121,323.831,353.988,170.316,51.434,160.046
C00642=1016.128,324.079,353.954,170.322,51.429,160.046
C00643=1016.136,324.327,353.920,170.330,51.425,160.046
C00644=1016.141,324.574,353.887,170.335,51.421,160.046
C00645=1016.148,324.822,353.853,170.343,51.416,160.047
C00646=1016.156,325.070,353.819,170.350,51.412,160.047
C00647=1016.162,325.317,353.786,170.356,51.408,160.047
C00648=1016.169,325.564,353.752,170.363,51.404,160.047
C00649=1016.176,325.812,353.717,170.370,51.399,160.048
C00650=1016.183,326.060,353.684,170.377,51.395,160.048
C00651=1016.189,326.307,353.650,170.383,51.391,160.048
C00652=1016.196,326.555,353.616,170.390,51.386,160.048
C00653=1016.203,326.803,353.581,170.396,51.383,160.049
C00654=1016.209,327.050,353.547,170.403,51.378,160.049
C00655=1016.216,327.297,353.513,170.411,51.374,160.049
C00656=1016.222,327.545,353.478,170.417,51.370,160.049
C00657=1016.229,327.793,353.444,170.424,51.366,160.050
C00658=1016.236,328.040,353.410,170.431,51.362,160.050
C00659=1016.242,328.288,353.375,170.437,51.358,160.050
C00660=1016.249,328.536,353.341,170.445,51.354,160.051
C00661=1016.256,328.783,353.306,170.452,51.350,160.051
C00662=1016.263,329.031,353.272,170.458,51.346,160.051
C00663=1016.269,329.278,353.237,170.465,51.342,160.051
C00664=1016.276,329.525,353.203,170.472,51.337,160.052
C00665=1016.283,329.773,353.169,170.479,51.334,160.052
C00666=1016.289,330.020,353.134,170.486,51.329,160.052
C00667=1016.297,330.268,353.100,170.493,51.325,160.053
C00668=1016.303,330.515,353.065,170.499,51.321,160.053
C00669=1016.310,330.763,353.030,170.507,51.318,160.053
C00670=1016.317,331.011,352.996,170.514,51.314,160.054
C00671=1016.324,331.258,352.961,170.520,51.310,160.054
C00672=1016.330,331.506,352.926,170.527,51.306,160.054
C00673=1016.337,331.753,352.891,170.535,51.301,160.054
C00674=1016.344,332.001,352.857,170.541,51.298,160.055
C00675=1016.351,332.248,352.822,170.548,51.294,160.055
C00676=1016.358,332.496,352.787,170.556,51.290,160.056
C00677=1016.364,332.744,352.753,170.562,51.287,160.056
C00678=1016.371,332.991,352.717,170.569,51.282,160.056
C00679=1016.378,333.238,352.682,170.577,51.278,160.057
C00680=1016.385,333.485,352.648,170.583,51.275,160.057
C00681=1016.392,333.733,352.613,170.590,51.271,160.057
C00682=1016.399,333.980,352.578,170.598,51.267,160.058
C00683=1016.406,334.227,352.542,170.604,51.263,160.058
C00684=1016.413,334.475,352.507,170.612,51.260,160.059
C00685=1016.419,334.722,352.472,170.619,51.256,160.059
C00686=1016.426,334.970,352.437,170.627,51.252,160.059
C00687=1016.433,335.217,352.402,170.633,51.248,160.060
C00688=1016.440,335.464,352.367,170.640,51.245,160.060
C00689=1016.447,335.712,352.331,170.648,51.241,160.060
C00690=1016.454,335.960,352.296,170.654,51.237,160.061
C00691=1016.461,336.207,352.261,170.662,51.234,160.061
C00692=1016.467,336.454,352.226,170.669,51.230,160.062
C00693=1016.474,336.702,352.191,170.676,51.226,160.062
C00694=1016.481,336.950,352.155,170.683,51.223,160.063
C00695=1016.488,337.197,352.120,170.690,51.219,160.063
C00696=1016.496,337.469,352.081,170.698,51.215,160.063
C00697=1016.504,337.740,352.042,170.706,51.211,160.064
C00698=1016.512,338.011,352.003,170.714,51.207,160.064
C00699=1016.519,338.283,351.965,170.722,51.203,160.065
C00700=1016.526,338.530,351.929,170.730,51.199,160.065
C00701=1016.534,338.778,351.894,170.736,51.196,160.066
C00702=1016.540,339.025,351.859,170.744,51.192,160.066
C00703=1016.547,339.272,351.823,170.751,51.189,160.067
C00704=1016.554,339.519,351.788,170.759,51.185,160.067
C00705=1016.561,339.767,351.751,170.766,51.182,160.068
C00706=1016.568,340.014,351.716,170.773,51.178,160.068
C00707=1016.575,340.261,351.680,170.781,51.175,160.069
C00708=1016.582,340.509,351.645,170.787,51.172,160.069
C00709=1016.589,340.756,351.609,170.795,51.168,160.070
C00710=1016.596,341.004,351.572,170.803,51.165,160.070
C00711=1016.603,341.251,351.537,170.810,51.161,160.071
C00712=1016.610,341.498,351.501,170.817,51.158,160.071
C00713=1016.618,341.746,351.465,170.824,51.154,160.072
C00714=1016.625,341.993,351.430,170.832,51.151,160.072
C00715=1016.632,342.240,351.393,170.840,51.147,160.073
C00716=1016.639,342.487,351.357,170.847,51.145,160.073
C00717=1016.646,342.735,351.321,170.854,51.141,160.074
C00718=1016.653,342.982,351.286,170.862,51.138,160.074
C00719=1016.660,343.230,351.249,170.869,51.134,160.075
C00720=1016.667,343.476,351.213,170.876,51.131,160.075
C00721=1016.675,343.724,351.177,170.884,51.128,160.076
C00722=1016.681,343.971,351.140,170.892,51.125,160.076
C00723=1016.688,344.219,351.105,170.899,51.121,160.077
C00724=1016.696,344.466,351.068,170.907,51.118,160.078
C00725=1016.703,344.713,351.033,170.914,51.115,160.078
C00726=1016.710,344.961,350.996,170.921,51.111,160.079
C00727=1016.717,345.208,350.960,170.929,51.109,160.079
C00728=1016.725,345.455,350.924,170.937,51.105,160.080
C00729=1016.732,345.703,350.887,170.945,51.102,160.081
C00730=1016.739,345.950,350.851,170.952,51.099,160.081
C00731=1016.747,346.196,350.814,170.959,51.095,160.082
C00732=1016.755,346.444,350.778,170.967,51.092,160.082
C00733=1016.761,346.691,350.741,170.975,51.089,160.083
C00734=1016.769,346.938,350.705,170.983,51.086,160.083
C00735=1016.776,347.186,350.668,170.991,51.083,160.084
C00736=1016.784,347.433,350.632,170.997,51.080,160.085
C00737=1016.790,347.680,350.595,171.005,51.077,160.085
C00738=1016.798,347.927,350.559,171.013,51.074,160.086
C00739=1016.805,348.175,350.521,171.021,51.071,160.087
C00740=1016.812,348.422,350.485,171.029,51.068,160.087
C00741=1016.819,348.668,350.448,171.037,51.065,160.088
C00742=1016.827,348.916,350.412,171.044,51.062,160.088
C00743=1016.834,349.164,350.375,171.052,51.059,160.089
C00744=1016.842,349.410,350.338,171.060,51.056,160.090
C00745=1016.849,349.658,350.301,171.068,51.053,160.091
C00746=1016.855,349.905,350.264,171.075,51.049,160.091
C00747=1016.863,350.151,350.227,171.083,51.047,160.092
C00748=1016.870,350.399,350.190,171.091,51.044,160.093
C00749=1016.878,350.646,350.153,171.098,51.041,160.093
C00750=1016.885,350.894,350.117,171.106,51.038,160.094
C00751=1016.893,351.141,350.080,171.114,51.035,160.095
C00752=1016.900,351.388,350.042,171.122,51.032,160.095
C00753=1016.908,351.635,350.006,171.130,51.030,160.096
C00754=1016.915,351.882,349.968,171.138,51.027,160.097
C00755=1016.923,352.130,349.931,171.146,51.024,160.097
C00756=1016.931,352.398,349.891,171.154,51.021,160.098
C00757=1016.940,352.667,349.850,171.163,51.018,160.099
C00758=1016.947,352.936,349.810,171.172,51.014,160.100
C00759=1016.955,353.204,349.770,171.180,51.011,160.101
C00760=1016.963,353.451,349.733,171.188,51.009,160.101
C00761=1016.971,353.698,349.695,171.196,51.006,160.102
C00762=1016.978,353.946,349.658,171.204,51.003,160.103
C00763=1016.985,354.193,349.620,171.213,51.001,160.104
C00764=1016.993,354.440,349.583,171.221,50.998,160.104
C00765=1017.000,354.687,349.546,171.229,50.995,160.105
C00766=1017.008,354.934,349.508,171.237,50.992,160.106
C00767=1017.015,355.180,349.470,171.245,50.990,160.107
C00768=1017.023,355.427,349.433,171.253,50.987,160.107
C00769=1017.030,355.674,349.395,171.261,50.984,160.108
C00770=1017.038,355.922,349.357,171.269,50.982,160.109
C00771=1017.046,356.169,349.320,171.277,50.979,160.110
C00772=1017.054,356.415,349.282,171.285,50.976,160.110
C00773=1017.061,356.663,349.245,171.294,50.973,160.111
C00774=1017.068,356.910,349.207,171.302,50.971,160.112
C00775=1017.076,357.158,349.169,171.310,50.968,160.113
C00776=1017.084,357.404,349.132,171.318,50.965,160.114
C00777=1017.092,357.651,349.094,171.327,50.963,160.115
C00778=1017.100,357.898,349.056,171.335,50.960,160.115
C00779=1017.107,358.145,349.018,171.343,50.958,160.116
C00780=1017.115,358.392,348.980,171.351,50.955,160.117
C00781=1017.122,358.640,348.942,171.359,50.953,160.118
C00782=1017.131,358.886,348.904,171.368,50.951,160.119
C00783=1017.138,359.133,348.867,171.376,50.948,160.120
C00784=1017.146,359.380,348.828,171.384,50.945,160.121
C00785=1017.154,359.627,348.790,171.393,50.943,160.121
C00786=1017.161,359.874,348.752,171.401,50.941,160.122
C00787=1017.168,360.121,348.713,171.409,50.938,160.123
C00788=1017.176,360.368,348.675,171.417,50.936,160.124
C00789=1017.183,360.614,348.637,171.426,50.933,160.125
C00790=1017.192,360.862,348.598,171.434,50.931,160.126
C00791=1017.199,361.108,348.560,171.443,50.929,160.127
C00792=1017.207,361.356,348.522,171.451,50.927,160.128
C00793=1017.215,361.602,348.484,171.459,50.924,160.129
C00794=1017.223,361.850,348.445,171.468,50.922,160.130
C00795=1017.230,362.096,348.407,171.476,50.920,160.130
C00796=1017.238,362.343,348.368,171.485,50.918,160.131
C00797=1017.246,362.590,348.330,171.494,50.915,160.132
C00798=1017.254,362.837,348.291,171.502,50.913,160.133
C00799=1017.261,363.084,348.252,171.511,50.910,160.134
C00800=1017.269,363.331,348.213,171.519,50.908,160.135
C00801=1017.278,363.578,348.175,171.528,50.906,160.136
C00802=1017.285,363.824,348.136,171.536,50.904,160.137
C00803=1017.293,364.071,348.098,171.544,50.901,160.138
C00804=1017.301,364.319,348.059,171.553,50.899,160.139
C00805=1017.309,364.565,348.021,171.563,50.897,160.140
C00806=1017.317,364.812,347.982,171.571,50.895,160.141
C00807=1017.326,365.059,347.943,171.579,50.892,160.142
C00808=1017.333,365.306,347.905,171.588,50.890,160.143
C00809=1017.342,365.552,347.865,171.597,50.889,160.144
C00810=1017.350,365.799,347.827,171.606,50.886,160.145
C00811=1017.357,366.047,347.788,171.614,50.884,160.146
C00812=1017.365,366.293,347.749,171.623,50.881,160.147
C00813=1017.373,366.540,347.710,171.632,50.880,160.148
C00814=1017.382,366.787,347.671,171.640,50.877,160.149
C00815=1017.390,367.034,347.632,171.650,50.875,160.150
C00816=1017.399,367.310,347.588,171.659,50.873,160.151
C00817=1017.408,367.586,347.544,171.669,50.871,160.152
C00818=1017.417,367.862,347.500,171.679,50.869,160.154
C00819=1017.425,368.138,347.456,171.690,50.866,160.155
C00820=1017.434,368.385,347.417,171.698,50.864,160.156
C00821=1017.442,368.632,347.378,171.707,50.863,160.157
C00822=1017.450,368.879,347.338,171.716,50.861,160.158
C00823=1017.458,369.125,347.299,171.725,50.858,160.159
C00824=1017.466,369.372,347.259,171.734,50.857,160.160
C00825=1017.474,369.618,347.220,171.742,50.855,160.161
C00826=1017.482,369.865,347.181,171.751,50.853,160.162
C00827=1017.490,370.112,347.141,171.761,50.851,160.163
C00828=1017.498,370.358,347.101,171.769,50.849,160.165
C00829=1017.506,370.605,347.061,171.778,50.847,160.166
C00830=1017.515,370.852,347.022,171.788,50.845,160.167
C00831=1017.522,371.099,346.982,171.797,50.844,160.168
C00832=1017.531,371.346,346.942,171.806,50.842,160.169
C00833=1017.540,371.593,346.903,171.815,50.839,160.170
C00834=1017.548,371.840,346.863,171.824,50.838,160.171
C00835=1017.556,372.086,346.823,171.833,50.836,160.172
C00836=1017.564,372.332,346.783,171.842,50.834,160.174
C00837=1017.573,372.579,346.744,171.851,50.832,160.175
C00838=1017.581,372.826,346.705,171.861,50.831,160.176
C00839=1017.589,373.072,346.664,171.870,50.829,160.177
C00840=1017.598,373.319,346.624,171.879,50.828,160.179
C00841=1017.606,373.566,346.584,171.889,50.826,160.180
C00842=1017.615,373.812,346.544,171.898,50.824,160.181
C00843=1017.622,374.059,346.504,171.907,50.822,160.182
C00844=1017.632,374.306,346.464,171.916,50.820,160.183
C00845=1017.640,374.552,346.425,171.926,50.819,160.185
C00846=1017.648,374.799,346.384,171.935,50.817,160.186
C00847=1017.657,375.045,346.345,171.945,50.815,160.187
C00848=1017.665,375.292,346.304,171.954,50.814,160.188
C00849=1017.674,375.538,346.264,171.964,50.812,160.190
C00850=1017.682,375.786,346.223,171.973,50.810,160.191
C00851=1017.691,376.032,346.183,171.982,50.808,160.192
C00852=1017.699,376.278,346.143,171.992,50.807,160.193
C00853=1017.708,376.525,346.102,172.000,50.806,160.194
C00854=1017.716,376.771,346.061,172.011,50.804,160.196
C00855=1017.725,377.017,346.021,172.020,50.803,160.197
C00856=1017.733,377.264,345.980,172.030,50.801,160.198
C00857=1017.741,377.510,345.939,172.040,50.800,160.200
C00858=1017.750,377.757,345.898,172.049,50.798,160.201
C00859=1017.758,378.004,345.858,172.059,50.797,160.202
C00860=1017.767,378.250,345.817,172.068,50.796,160.204
C00861=1017.775,378.497,345.777,172.078,50.794,160.205
C00862=1017.784,378.744,345.736,172.087,50.793,160.206
C00863=1017.792,378.990,345.695,172.097,50.791,160.208
C00864=1017.801,379.237,345.655,172.107,50.790,160.209
C00865=1017.810,379.482,345.613,172.116,50.789,160.210
C00866=1017.818,379.729,345.572,172.126,50.787,160.212
C00867=1017.827,379.976,345.531,172.135,50.786,160.213
C00868=1017.836,380.222,345.491,172.146,50.784,160.214
C00869=1017.845,380.469,345.450,172.156,50.783,160.216
C00870=1017.853,380.715,345.409,172.165,50.782,160.217
C00871=1017.861,380.961,345.367,172.175,50.780,160.219
C00872=1017.871,381.208,345.327,172.185,50.779,160.220
C00873=1017.880,381.454,345.285,172.194,50.778,160.221
C00874=1017.888,381.701,345.244,172.205,50.776,160.223
C00875=1017.897,381.947,345.203,172.215,50.775,160.224
C00876=1017.907,382.246,345.153,172.226,50.774,160.226
C00877=1017.918,382.545,345.103,172.239,50.772,160.228
C00878=1017.929,382.843,345.053,172.251,50.770,160.229
C00879=1017.940,383.142,345.004,172.263,50.769,160.231
C00880=1017.949,383.388,344.962,172.273,50.768,160.233
C00881=1017.958,383.634,344.921,172.283,50.767,160.234
C00882=1017.967,383.880,344.879,172.294,50.765,160.236
C00883=1017.976,384.127,344.838,172.303,50.764,160.237
C00884=1017.985,384.374,344.796,172.313,50.763,160.239
C00885=1017.994,384.620,344.755,172.324,50.762,160.240
C00886=1018.003,384.866,344.714,172.334,50.760,160.241
C00887=1018.012,385.113,344.672,172.344,50.760,160.243
C00888=1018.021,385.359,344.630,172.355,50.758,160.244
C00889=1018.030,385.605,344.588,172.365,50.757,160.246
C00890=1018.039,385.852,344.547,172.374,50.756,160.247
C00891=1018.048,386.098,344.505,172.385,50.756,160.249
C00892=1018.057,386.344,344.462,172.395,50.755,160.251
C00893=1018.066,386.590,344.421,172.406,50.753,160.252
C00894=1018.075,386.836,344.379,172.416,50.752,160.254
C00895=1018.084,387.083,344.337,172.427,50.752,160.255
C00896=1018.093,387.329,344.295,172.437,50.750,160.257
C00897=1018.102,387.575,344.253,172.447,50.749,160.259
C00898=1018.112,387.821,344.210,172.458,50.748,160.260
C00899=1018.121,388.068,344.169,172.469,50.748,160.262
C00900=1018.130,388.313,344.126,172.479,50.747,160.263
C00901=1018.138,388.560,344.084,172.490,50.746,160.265
C00902=1018.148,388.806,344.042,172.500,50.745,160.267
C00903=1018.157,389.053,343.999,172.511,50.744,160.268
C00904=1018.166,389.299,343.957,172.521,50.743,160.270
C00905=1018.176,389.544,343.915,172.532,50.742,160.271
C00906=1018.184,389.791,343.872,172.543,50.742,160.273
C00907=1018.194,390.038,343.829,172.553,50.741,160.275
C00908=1018.203,390.283,343.787,172.564,50.740,160.277
C00909=1018.212,390.529,343.745,172.574,50.739,160.278
C00910=1018.222,390.776,343.702,172.585,50.738,160.280
C00911=1018.231,391.021,343.659,172.596,50.737,160.281
C00912=1018.240,391.268,343.616,172.606,50.737,160.283
C00913=1018.250,391.514,343.574,172.617,50.736,160.285
C00914=1018.259,391.760,343.531,172.629,50.735,160.287
C00915=1018.269,392.006,343.488,172.639,50.734,160.288
C00916=1018.278,392.252,343.446,172.650,50.734,160.290
C00917=1018.287,392.498,343.402,172.661,50.733,160.292
C00918=1018.296,392.744,343.360,172.672,50.733,160.294
C00919=1018.306,392.991,343.317,172.682,50.732,160.295
C00920=1018.315,393.236,343.274,172.694,50.731,160.297
C00921=1018.325,393.483,343.231,172.705,50.731,160.299
C00922=1018.335,393.729,343.188,172.716,50.730,160.301
C00923=1018.343,393.974,343.144,172.726,50.729,160.302
C00924=1018.353,394.221,343.101,172.738,50.729,160.304
C00925=1018.363,394.466,343.058,172.749,50.728,160.306
C00926=1018.372,394.713,343.015,172.760,50.728,160.308
C00927=1018.382,394.959,342.971,172.772,50.727,160.310
C00928=1018.391,395.204,342.929,172.783,50.727,160.312
C00929=1018.401,395.450,342.885,172.793,50.726,160.313
C00930=1018.411,395.696,342.841,172.805,50.725,160.315
C00931=1018.421,395.943,342.798,172.816,50.725,160.317
C00932=1018.430,396.189,342.754,172.827,50.725,160.319
C00933=1018.440,396.434,342.711,172.839,50.724,160.321
C00934=1018.449,396.680,342.667,172.850,50.724,160.323
C00935=1018.459,396.927,342.624,172.861,50.724,160.325
C00936=1018.472,397.263,342.564,172.877,50.723,160.327
C00937=1018.486,397.599,342.504,172.893,50.723,160.330
C00938=1018.499,397.935,342.444,172.908,50.722,160.332
C00939=1018.512,398.271,342.384,172.924,50.721,160.335
C00940=1018.522,398.517,342.341,172.936,50.721,160.337
C00941=1018.532,398.763,342.297,172.947,50.720,160.339
C00942=1018.542,399.009,342.253,172.959,50.720,160.341
C00943=1018.551,399.255,342.209,172.970,50.720,160.343
C00944=1018.561,399.501,342.164,172.982,50.719,160.345
C00945=1018.571,399.747,342.121,172.993,50.719,160.347
C00946=1018.581,399.992,342.076,173.006,50.719,160.349
C00947=1018.591,400.239,342.032,173.018,50.718,160.351
C00948=1018.601,400.485,341.988,173.029,50.719,160.353
C00949=1018.611,400.730,341.943,173.041,50.718,160.355
C00950=1018.621,400.976,341.899,173.052,50.718,160.357
C00951=1018.630,401.222,341.855,173.065,50.718,160.359
C00952=1018.640,401.467,341.810,173.077,50.718,160.361
C00953=1018.650,401.713,341.765,173.088,50.718,160.363
C00954=1018.661,401.959,341.721,173.100,50.718,160.365
C00955=1018.670,402.205,341.677,173.112,50.717,160.367
C00956=1018.680,402.450,341.632,173.124,50.717,160.369
C00957=1018.690,402.696,341.587,173.136,50.717,160.371
C00958=1018.701,402.942,341.542,173.148,50.717,160.373
C00959=1018.711,403.187,341.498,173.161,50.717,160.376
C00960=1018.720,403.433,341.453,173.172,50.718,160.378
C00961=1018.731,403.679,341.408,173.184,50.717,160.380
C00962=1018.741,403.924,341.363,173.197,50.717,160.382
C00963=1018.751,404.170,341.318,173.209,50.717,160.384
C00964=1018.761,404.416,341.273,173.221,50.717,160.386
C00965=1018.771,404.661,341.228,173.234,50.717,160.388
C00966=1018.782,404.907,341.184,173.245,50.717,160.390
C00967=1018.792,405.153,341.138,173.258,50.717,160.393
C00968=1018.802,405.398,341.093,173.270,50.717,160.395
C00969=1018.812,405.645,341.048,173.283,50.718,160.397
C00970=1018.823,405.889,341.003,173.295,50.717,160.399
C00971=1018.834,406.135,340.958,173.307,50.717,160.401
C00972=1018.844,406.382,340.913,173.320,50.717,160.404
C00973=1018.855,406.626,340.868,173.332,50.718,160.406
C00974=1018.865,406.872,340.822,173.345,50.718,160.408
C00975=1018.876,407.118,340.777,173.358,50.718,160.410
C00976=1018.885,407.364,340.732,173.370,50.718,160.413
C00977=1018.897,407.609,340.686,173.383,50.718,160.415
C00978=1018.907,407.854,340.641,173.396,50.718,160.417
C00979=1018.918,408.101,340.595,173.409,50.718,160.420
C00980=1018.928,408.346,340.549,173.422,50.719,160.422
C00981=1018.939,408.592,340.504,173.434,50.719,160.424
C00982=1018.950,408.837,340.458,173.447,50.719,160.426
C00983=1018.960,409.083,340.412,173.459,50.720,160.429
C00984=1018.970,409.328,340.366,173.472,50.720,160.431
C00985=1018.981,409.573,340.320,173.485,50.720,160.433
C00986=1018.991,409.819,340.274,173.498,50.720,160.436
C00987=1019.002,410.065,340.228,173.511,50.720,160.438
C00988=1019.013,410.310,340.183,173.524,50.721,160.441
C00989=1019.024,410.555,340.136,173.537,50.721,160.443
C00990=1019.034,410.801,340.090,173.550,50.721,160.445
C00991=1019.045,411.046,340.044,173.563,50.722,160.448
C00992=1019.055,411.292,339.998,173.577,50.723,160.450
C00993=1019.067,411.538,339.951,173.590,50.723,160.453
C00994=1019.078,411.783,339.905,173.603,50.723,160.455
C00995=1019.088,412.028,339.859,173.616,50.723,160.458
C00996=1019.104,412.387,339.791,173.636,50.724,160.461
C00997=1019.120,412.745,339.723,173.655,50.725,160.465
C00998=1019.136,413.104,339.655,173.674,50.726,160.469
C00999=1019.152,413.462,339.587,173.695,50.727,160.472
C01000=1019.164,413.708,339.540,173.707,50.727,160.475
C01001=1019.175,413.953,339.494,173.722,50.728,160.477
C01002=1019.185,414.198,339.447,173.734,50.728,160.480
C01003=1019.196,414.444,339.400,173.748,50.729,160.482
C01004=1019.207,414.689,339.354,173.763,50.729,160.485
C01005=1019.218,414.935,339.307,173.776,50.730,160.488
C01006=1019.229,415.180,339.260,173.789,50.730,160.490
C01007=1019.240,415.425,339.212,173.804,50.731,160.493
C01008=1019.255,415.744,339.151,173.821,50.733,160.496
C01009=1019.269,416.063,339.090,173.839,50.733,160.500
C01010=1019.284,416.381,339.028,173.857,50.734,160.503
C01011=1019.298,416.700,338.967,173.875,50.735,160.507
C01012=1019.309,416.946,338.920,173.889,50.736,160.509
C01013=1019.321,417.191,338.872,173.903,50.736,160.512
C01014=1019.332,417.436,338.824,173.917,50.737,160.515
C01015=1019.343,417.681,338.777,173.932,50.738,160.518
C01016=1019.355,417.926,338.729,173.945,50.739,160.520
C01017=1019.367,418.172,338.682,173.959,50.740,160.523
C01018=1019.377,418.417,338.634,173.974,50.741,160.526
C01019=1019.389,418.662,338.587,173.988,50.741,160.528
C01020=1019.018,416.680,338.631,173.860,50.805,160.524
C01021=1019.006,416.435,338.679,173.846,50.805,160.521
C01022=1018.995,416.190,338.726,173.832,50.804,160.519
C01023=1018.984,415.944,338.773,173.819,50.803,160.516
C01024=1018.973,415.700,338.821,173.805,50.802,160.513
C01025=1018.962,415.454,338.868,173.791,50.802,160.511
C01026=1018.951,415.209,338.915,173.776,50.801,160.508
C01027=1018.940,414.963,338.962,173.764,50.801,160.506
C01028=1018.929,414.718,339.009,173.750,50.800,160.503
C01029=1018.917,414.473,339.056,173.735,50.800,160.500
C01030=1018.907,414.228,339.102,173.722,50.800,160.498
C01031=1018.895,413.982,339.149,173.709,50.799,160.495
C01032=1018.884,413.737,339.196,173.695,50.799,160.493
C01033=1018.866,413.334,339.272,173.673,50.798,160.489
C01034=1018.848,412.930,339.349,173.650,50.797,160.484
C01035=1018.830,412.527,339.425,173.629,50.797,160.480
C01036=1018.812,412.123,339.501,173.607,50.796,160.476
C01037=1018.802,411.877,339.548,173.593,50.796,160.474
C01038=1018.791,411.632,339.594,173.580,50.795,160.471
C01039=1018.781,411.387,339.640,173.567,50.795,160.469
C01040=1018.770,411.142,339.687,173.554,50.795,160.467
C01041=1018.759,410.896,339.733,173.541,50.795,160.464
C01042=1018.748,410.651,339.779,173.527,50.795,160.462
C01043=1018.738,410.405,339.825,173.515,50.794,160.459
C01044=1018.727,410.160,339.871,173.501,50.794,160.457
C01045=1018.716,409.914,339.917,173.488,50.794,160.455
C01046=1018.706,409.669,339.963,173.475,50.793,160.452
C01047=1018.695,409.423,340.009,173.463,50.793,160.450
C01048=1018.684,409.178,340.055,173.449,50.793,160.448
C01049=1018.674,408.932,340.101,173.436,50.793,160.445
C01050=1018.663,408.686,340.147,173.424,50.792,160.443
C01051=1018.652,408.441,340.193,173.411,50.793,160.441
C01052=1018.642,408.195,340.238,173.398,50.792,160.438
C01053=1018.632,407.955,340.283,173.385,50.793,160.436
C01054=1018.621,407.715,340.327,173.372,50.792,160.434
C01055=1018.611,407.474,340.371,173.360,50.792,160.431
C01056=1018.600,407.234,340.415,173.349,50.792,160.429
C01057=1018.591,406.994,340.460,173.336,50.792,160.427
C01058=1018.580,406.754,340.505,173.324,50.792,160.425
C01059=1018.569,406.514,340.549,173.311,50.792,160.423
C01060=1018.560,406.274,340.593,173.299,50.792,160.421
C01061=1018.549,406.027,340.638,173.287,50.792,160.418
C01062=1018.539,405.782,340.682,173.274,50.792,160.416
C01063=1018.528,405.536,340.728,173.262,50.792,160.414
C01064=1018.519,405.291,340.773,173.249,50.792,160.412
C01065=1018.508,405.045,340.818,173.237,50.793,160.410
C01066=1018.498,404.800,340.863,173.225,50.793,160.408
C01067=1018.487,404.554,340.909,173.212,50.793,160.405
C01068=1018.477,404.308,340.953,173.200,50.793,160.403
C01069=1018.466,404.063,340.998,173.188,50.793,160.401
C01070=1018.457,403.817,341.043,173.175,50.793,160.399
C01071=1018.447,403.572,341.088,173.163,50.793,160.397
C01072=1018.437,403.325,341.133,173.151,50.793,160.395
C01073=1018.426,403.080,341.177,173.138,50.793,160.392
C01074=1018.417,402.835,341.222,173.127,50.794,160.391
C01075=1018.406,402.588,341.267,173.115,50.794,160.388
C01076=1018.397,402.342,341.311,173.102,50.794,160.386
C01077=1018.386,402.097,341.355,173.091,50.795,160.384
C01078=1018.376,401.851,341.401,173.078,50.795,160.382
C01079=1018.366,401.605,341.445,173.067,50.794,160.380
C01080=1018.356,401.359,341.489,173.055,50.795,160.378
C01081=1018.346,401.114,341.534,173.042,50.795,160.376
C01082=1018.337,400.868,341.579,173.031,50.796,160.374
C01083=1018.327,400.622,341.623,173.019,50.796,160.372
C01084=1018.317,400.377,341.667,173.007,50.796,160.370
C01085=1018.307,400.131,341.711,172.995,50.797,160.368
C01086=1018.297,399.884,341.755,172.984,50.797,160.366
C01087=1018.287,399.639,341.800,172.972,50.797,160.364
C01088=1018.278,399.393,341.844,172.960,50.798,160.362
C01089=1018.267,399.147,341.887,172.949,50.798,160.360
C01090=1018.258,398.901,341.932,172.937,50.798,160.358
C01091=1018.248,398.656,341.976,172.926,50.799,160.356
C01092=1018.238,398.410,342.020,172.914,50.799,160.354
C01093=1018.225,398.060,342.081,172.897,50.800,160.352
C01094=1018.211,397.711,342.144,172.881,50.801,160.349
C01095=1018.197,397.361,342.206,172.864,50.802,160.346
C01096=1018.183,397.012,342.268,172.849,50.802,160.344
C01097=1018.173,396.766,342.312,172.837,50.803,160.342
C01098=1018.163,396.520,342.355,172.826,50.803,160.340
C01099=1018.155,396.274,342.399,172.814,50.804,160.338
C01100=1018.144,396.028,342.442,172.803,50.805,160.336
C01101=1018.135,395.782,342.485,172.791,50.806,160.334
C01102=1018.125,395.536,342.529,172.780,50.806,160.332
C01103=1018.116,395.291,342.572,172.769,50.806,160.331
C01104=1018.106,395.044,342.615,172.758,50.807,160.329
C01105=1018.096,394.798,342.659,172.747,50.808,160.327
C01106=1018.087,394.552,342.702,172.735,50.809,160.325
C01107=1018.077,394.306,342.745,172.724,50.809,160.323
C01108=1018.068,394.060,342.789,172.714,50.810,160.322
C01109=1018.059,393.814,342.831,172.702,50.811,160.320
C01110=1018.049,393.568,342.875,172.691,50.812,160.318
C01111=1018.040,393.322,342.918,172.680,50.812,160.316
C01112=1018.030,393.076,342.960,172.668,50.813,160.315
C01113=1018.021,392.830,343.004,172.658,50.814,160.313
C01114=1018.012,392.584,343.047,172.647,50.814,160.311
C01115=1018.002,392.338,343.089,172.636,50.815,160.309
C01116=1017.992,392.092,343.132,172.625,50.816,160.308
C01117=1017.983,391.846,343.175,172.614,50.817,160.306
C01118=1017.974,391.599,343.218,172.603,50.817,160.304
C01119=1017.965,391.353,343.261,172.593,50.818,160.302
C01120=1017.955,391.107,343.303,172.582,50.819,160.301
C01121=1017.946,390.861,343.346,172.570,50.820,160.299
C01122=1017.937,390.615,343.388,172.560,50.821,160.297
C01123=1017.927,390.369,343.431,172.549,50.822,160.296
C01124=1017.918,390.123,343.474,172.539,50.823,160.294
C01125=1017.909,389.877,343.516,172.528,50.824,160.293
C01126=1017.899,389.630,343.559,172.518,50.825,160.291
C01127=1017.890,389.384,343.601,172.506,50.826,160.289
C01128=1017.881,389.138,343.643,172.495,50.827,160.288
C01129=1017.872,388.892,343.685,172.485,50.828,160.286
C01130=1017.863,388.645,343.728,172.474,50.828,160.284
C01131=1017.854,388.399,343.770,172.464,50.830,160.283
C01132=1017.845,388.153,343.813,172.454,50.831,160.281
C01133=1017.836,387.907,343.854,172.443,50.832,160.280
C01134=1017.827,387.661,343.897,172.433,50.833,160.278
C01135=1017.818,387.415,343.938,172.422,50.834,160.276
C01136=1017.808,387.168,343.981,172.412,50.835,160.275
C01137=1017.799,386.921,344.022,172.401,50.836,160.273
C01138=1017.790,386.676,344.065,172.391,50.837,160.272
C01139=1017.781,386.429,344.106,172.381,50.839,160.270
C01140=1017.772,386.183,344.148,172.370,50.839,160.269
C01141=1017.763,385.937,344.190,172.360,50.841,160.267
C01142=1017.754,385.690,344.232,172.349,50.842,160.266
C01143=1017.745,385.445,344.274,172.339,50.843,160.264
C01144=1017.736,385.198,344.316,172.329,50.844,160.262
C01145=1017.727,384.952,344.357,172.318,50.845,160.261
C01146=1017.718,384.705,344.399,172.308,50.847,160.260
C01147=1017.710,384.458,344.440,172.298,50.848,160.258
C01148=1017.700,384.212,344.481,172.287,50.849,160.257
C01149=1017.691,383.966,344.523,172.277,50.851,160.255
C01150=1017.682,383.720,344.565,172.268,50.852,160.254
C01151=1017.674,383.473,344.605,172.258,50.853,160.252
C01152=1017.664,383.227,344.646,172.248,50.855,160.251
C01153=1017.653,382.927,344.697,172.235,50.856,160.249
C01154=1017.642,382.625,344.747,172.223,50.858,160.247
C01155=1017.631,382.324,344.798,172.210,50.859,160.245
C01156=1017.621,382.023,344.848,172.199,50.861,160.244
C01157=1017.612,381.777,344.890,172.189,50.863,160.242
C01158=1017.604,381.531,344.930,172.178,50.864,160.241
C01159=1017.594,381.284,344.972,172.168,50.865,160.240
C01160=1017.586,381.037,345.013,172.158,50.867,160.238
C01161=1017.577,380.792,345.054,172.149,50.868,160.237
C01162=1017.569,380.545,345.095,172.139,50.869,160.235
C01163=1017.559,380.298,345.135,172.129,50.871,160.234
C01164=1017.551,380.052,345.177,172.119,50.873,160.233
C01165=1017.542,379.806,345.218,172.110,50.874,160.231
C01166=1017.534,379.559,345.258,172.099,50.875,160.230
C01167=1017.526,379.312,345.299,172.090,50.877,160.229
C01168=1017.516,379.066,345.340,172.080,50.878,160.227
C01169=1017.508,378.820,345.381,172.070,50.880,160.226
C01170=1017.499,378.573,345.422,172.060,50.882,160.225
C01171=1017.491,378.327,345.463,172.051,50.883,160.223
C01172=1017.482,378.080,345.503,172.041,50.885,160.222
C01173=1017.474,377.834,345.544,172.031,50.886,160.221
C01174=1017.466,377.587,345.584,172.022,50.888,160.220
C01175=1017.457,377.340,345.625,172.012,50.890,160.218
C01176=1017.448,377.094,345.665,172.003,50.891,160.217
C01177=1017.440,376.847,345.706,171.993,50.893,160.216
C01178=1017.432,376.601,345.747,171.983,50.895,160.214
C01179=1017.424,376.355,345.788,171.974,50.896,160.213
C01180=1017.414,376.108,345.828,171.965,50.898,160.212
C01181=1017.407,375.861,345.868,171.956,50.899,160.211
C01182=1017.399,375.615,345.909,171.946,50.901,160.209
C01183=1017.389,375.368,345.949,171.937,50.903,160.208
C01184=1017.382,375.121,345.989,171.927,50.905,160.207
C01185=1017.373,374.875,346.029,171.917,50.907,160.206
C01186=1017.364,374.628,346.069,171.908,50.908,160.205
C01187=1017.356,374.382,346.109,171.899,50.910,160.203
C01188=1017.347,374.135,346.149,171.889,50.911,160.202
C01189=1017.339,373.889,346.189,171.880,50.913,160.201
C01190=1017.330,373.642,346.229,171.871,50.915,160.200
C01191=1017.322,373.395,346.269,171.861,50.917,160.198
C01192=1017.314,373.149,346.309,171.852,50.919,160.197
C01193=1017.305,372.902,346.348,171.842,50.921,160.196
C01194=1017.298,372.655,346.388,171.834,50.923,160.195
C01195=1017.288,372.409,346.429,171.824,50.925,160.194
C01196=1017.280,372.162,346.469,171.815,50.927,160.193
C01197=1017.272,371.915,346.508,171.806,50.929,160.192
C01198=1017.264,371.669,346.547,171.797,50.931,160.190
C01199=1017.256,371.422,346.587,171.787,50.933,160.189
C01200=1017.247,371.175,346.626,171.778,50.934,160.188
C01201=1017.240,370.928,346.666,171.770,50.937,160.187
C01202=1017.231,370.682,346.706,171.760,50.939,160.186
C01203=1017.223,370.435,346.745,171.751,50.940,160.185
C01204=1017.215,370.188,346.785,171.742,50.942,160.183
C01205=1017.207,369.941,346.824,171.733,50.945,160.183
C01206=1017.199,369.695,346.864,171.724,50.946,160.181
C01207=1017.190,369.448,346.903,171.715,50.948,160.180
C01208=1017.183,369.201,346.943,171.706,50.951,160.179
C01209=1017.174,368.954,346.983,171.697,50.952,160.178
C01210=1017.166,368.709,347.022,171.688,50.955,160.177
C01211=1017.159,368.462,347.062,171.679,50.957,160.176
C01212=1017.150,368.214,347.100,171.671,50.959,160.175
C01213=1017.142,367.936,347.145,171.660,50.961,160.174
C01214=1017.133,367.657,347.190,171.650,50.963,160.173
C01215=1017.123,367.379,347.234,171.640,50.966,160.171
C01216=1017.114,367.100,347.278,171.630,50.968,160.170
C01217=1017.107,366.854,347.317,171.622,50.971,160.169
C01218=1017.098,366.607,347.356,171.612,50.973,160.168
C01219=1017.090,366.360,347.395,171.603,50.975,160.167
C01220=1017.082,366.113,347.433,171.595,50.977,160.166
C01221=1017.074,365.866,347.472,171.586,50.980,160.165
C01222=1017.066,365.620,347.511,171.577,50.982,160.164
C01223=1017.058,365.373,347.550,171.568,50.984,160.163
C01224=1017.050,365.126,347.588,171.560,50.986,160.162
C01225=1017.042,364.880,347.627,171.551,50.989,160.161
C01226=1017.033,364.632,347.666,171.542,50.991,160.160
C01227=1017.025,364.385,347.704,171.534,50.993,160.159
C01228=1017.018,364.139,347.743,171.525,50.996,160.158
C01229=1017.010,363.891,347.782,171.516,50.998,160.157
C01230=1017.002,363.645,347.821,171.508,51.000,160.156
C01231=1016.994,363.398,347.859,171.499,51.003,160.156
C01232=1016.986,363.151,347.898,171.491,51.005,160.155
C01233=1016.979,362.904,347.936,171.481,51.008,160.154
C01234=1016.971,362.657,347.975,171.473,51.010,160.153
C01235=1016.963,362.411,348.013,171.465,51.012,160.152
C01236=1016.955,362.163,348.052,171.456,51.015,160.151
C01237=1016.947,361.917,348.090,171.448,51.017,160.150
C01238=1016.939,361.670,348.129,171.440,51.020,160.149
C01239=1016.932,361.423,348.167,171.430,51.022,160.148
C01240=1016.924,361.175,348.205,171.422,51.025,160.147
C01241=1016.916,360.929,348.243,171.414,51.027,160.146
C01242=1016.909,360.681,348.282,171.405,51.029,160.145
C01243=1016.901,360.435,348.320,171.397,51.032,160.145
C01244=1016.894,360.188,348.359,171.389,51.034,160.144
C01245=1016.886,359.940,348.397,171.380,51.037,160.143
C01246=1016.878,359.694,348.435,171.372,51.040,160.142
C01247=1016.871,359.447,348.473,171.363,51.042,160.141
C01248=1016.863,359.200,348.512,171.355,51.045,160.140
C01249=1016.855,358.953,348.549,171.347,51.047,160.139
C01250=1016.848,358.707,348.587,171.338,51.050,160.138
C01251=1016.840,358.459,348.625,171.330,51.053,160.138
C01252=1016.832,358.212,348.663,171.322,51.055,160.137
C01253=1016.824,357.965,348.701,171.314,51.058,160.136
C01254=1016.817,357.717,348.738,171.305,51.060,160.135
C01255=1016.809,357.471,348.777,171.297,51.063,160.134
C01256=1016.802,357.224,348.814,171.288,51.066,160.134
C01257=1016.794,356.977,348.851,171.280,51.069,160.133
C01258=1016.786,356.730,348.890,171.272,51.071,160.132
C01259=1016.778,356.483,348.927,171.264,51.074,160.131
C01260=1016.771,356.236,348.965,171.256,51.077,160.130
C01261=1016.763,355.989,349.002,171.248,51.080,160.130
C01262=1016.756,355.742,349.040,171.240,51.082,160.129
C01263=1016.748,355.495,349.077,171.232,51.085,160.128
C01264=1016.741,355.247,349.115,171.223,51.088,160.127
C01265=1016.733,355.000,349.152,171.215,51.091,160.127
C01266=1016.725,354.753,349.190,171.207,51.094,160.126
C01267=1016.718,354.506,349.227,171.199,51.096,160.125
C01268=1016.711,354.259,349.265,171.191,51.099,160.124
C01269=1016.703,354.012,349.302,171.183,51.102,160.124
C01270=1016.696,353.765,349.339,171.175,51.105,160.123
C01271=1016.688,353.518,349.377,171.167,51.107,160.122
C01272=1016.681,353.271,349.414,171.159,51.110,160.121
C01273=1016.672,353.000,349.455,171.150,51.114,160.120
C01274=1016.665,352.729,349.495,171.141,51.118,160.120
C01275=1016.656,352.458,349.537,171.132,51.121,160.119
C01276=1016.647,352.187,349.577,171.124,51.124,160.118
C01277=1016.640,351.940,349.614,171.116,51.127,160.118
C01278=1016.632,351.693,349.651,171.108,51.130,160.117
C01279=1016.625,351.446,349.688,171.100,51.132,160.116
C01280=1016.618,351.198,349.725,171.092,51.135,160.115
C01281=1016.610,350.951,349.762,171.085,51.139,160.115
C01282=1016.603,350.705,349.799,171.077,51.142,160.114
C01283=1016.596,350.457,349.836,171.069,51.145,160.113
C01284=1016.589,350.210,349.873,171.061,51.148,160.113
C01285=1016.581,349.963,349.909,171.053,51.151,160.112
C01286=1016.574,349.715,349.947,171.045,51.154,160.112
C01287=1016.566,349.468,349.983,171.037,51.157,160.111
C01288=1016.560,349.222,350.020,171.029,51.160,160.110
C01289=1016.552,348.974,350.056,171.022,51.163,160.110
C01290=1016.545,348.727,350.094,171.013,51.166,160.109
C01291=1016.537,348.480,350.130,171.006,51.170,160.108
C01292=1016.530,348.232,350.168,170.998,51.173,160.108
C01293=1016.523,347.985,350.204,170.990,51.176,160.107
C01294=1016.516,347.738,350.240,170.982,51.179,160.106
C01295=1016.509,347.490,350.277,170.975,51.182,160.106
C01296=1016.501,347.244,350.314,170.968,51.185,160.105
C01297=1016.494,346.997,350.350,170.960,51.188,160.104
C01298=1016.487,346.749,350.387,170.952,51.192,160.104
C01299=1016.480,346.502,350.423,170.945,51.195,160.103
C01300=1016.473,346.254,350.459,170.937,51.198,160.103
C01301=1016.465,346.008,350.496,170.929,51.202,160.102
C01302=1016.458,345.761,350.532,170.921,51.205,160.102
C01303=1016.450,345.513,350.568,170.913,51.208,160.101
C01304=1016.443,345.266,350.605,170.906,51.212,160.100
C01305=1016.436,345.019,350.641,170.898,51.215,160.100
C01306=1016.429,344.771,350.677,170.891,51.218,160.099
C01307=1016.422,344.524,350.713,170.884,51.222,160.099
C01308=1016.415,344.276,350.749,170.876,51.225,160.098
C01309=1016.407,344.029,350.785,170.868,51.229,160.098
C01310=1016.401,343.782,350.822,170.861,51.232,160.097
C01311=1016.393,343.534,350.858,170.853,51.235,160.096
C01312=1016.386,343.288,350.894,170.845,51.239,160.096
C01313=1016.378,343.040,350.930,170.839,51.242,160.096
C01314=1016.372,342.792,350.966,170.831,51.245,160.095
C01315=1016.364,342.545,351.002,170.823,51.249,160.095
C01316=1016.357,342.298,351.038,170.816,51.253,160.094
C01317=1016.351,342.051,351.073,170.808,51.256,160.093
C01318=1016.344,341.803,351.110,170.801,51.260,160.093
C01319=1016.337,341.556,351.146,170.793,51.263,160.092
C01320=1016.329,341.308,351.181,170.786,51.266,160.092
C01321=1016.322,341.062,351.217,170.779,51.270,160.092
C01322=1016.315,340.814,351.252,170.771,51.274,160.091
C01323=1016.308,340.566,351.289,170.764,51.277,160.090
C01324=1016.301,340.320,351.325,170.756,51.281,160.090
C01325=1016.294,340.072,351.360,170.748,51.284,160.089
C01326=1016.287,339.825,351.396,170.742,51.288,160.089
C01327=1016.280,339.578,351.431,170.735,51.292,160.089
C01328=1016.274,339.329,351.468,170.727,51.295,160.088
C01329=1016.266,339.082,351.503,170.719,51.299,160.088
C01330=1016.260,338.835,351.539,170.712,51.302,160.087
C01331=1016.253,338.588,351.574,170.706,51.306,160.087
C01332=1016.245,338.340,351.610,170.698,51.310,160.086
C01333=1016.238,338.067,351.648,170.689,51.314,160.086
C01334=1016.230,337.793,351.688,170.681,51.318,160.085
C01335=1016.222,337.519,351.727,170.674,51.322,160.085
C01336=1016.215,337.245,351.766,170.665,51.326,160.084
C01337=1016.208,336.998,351.801,170.658,51.330,160.084
C01338=1016.200,336.751,351.836,170.651,51.334,160.084
C01339=1016.193,336.504,351.872,170.644,51.337,160.083
C01340=1016.186,336.257,351.907,170.637,51.341,160.083
C01341=1016.179,336.009,351.942,170.629,51.345,160.082
C01342=1016.172,335.761,351.977,170.622,51.349,160.082
C01343=1016.166,335.514,352.012,170.615,51.352,160.082
C01344=1016.159,335.267,352.048,170.608,51.357,160.081
C01345=1016.152,335.019,352.083,170.601,51.360,160.081
C01346=1016.145,334.772,352.118,170.594,51.364,160.080
C01347=1016.139,334.524,352.152,170.586,51.369,160.080
C01348=1016.132,334.276,352.187,170.580,51.372,160.080
C01349=1016.125,334.029,352.223,170.573,51.376,160.079
C01350=1016.119,333.782,352.258,170.565,51.380,160.079
C01351=1016.112,333.534,352.293,170.558,51.384,160.079
C01352=1016.105,333.287,352.328,170.552,51.388,160.078
C01353=1016.098,333.040,352.363,170.544,51.392,160.078
C01354=1016.091,332.792,352.397,170.537,51.395,160.078
C01355=1016.084,332.545,352.432,170.530,51.400,160.077
C01356=1016.077,332.297,352.467,170.523,51.404,160.077
C01357=1016.071,332.049,352.502,170.516,51.408,160.077
C01358=1016.064,331.802,352.537,170.509,51.412,160.076
C01359=1016.057,331.555,352.571,170.501,51.416,160.076
C01360=1016.050,331.307,352.606,170.494,51.420,160.076
C01361=1016.044,331.059,352.641,170.488,51.424,160.075
C01362=1016.036,330.812,352.675,170.481,51.428,160.075
C01363=1016.030,330.564,352.710,170.474,51.432,160.075
C01364=1016.023,330.316,352.744,170.466,51.436,160.074
C01365=1016.016,330.069,352.779,170.460,51.440,160.074
C01366=1016.009,329.821,352.813,170.453,51.444,160.074
C01367=1016.003,329.574,352.847,170.446,51.449,160.074
C01368=1015.996,329.327,352.882,170.439,51.453,160.073
C01369=1015.989,329.079,352.916,170.433,51.457,160.073
C01370=1015.983,328.832,352.951,170.425,51.461,160.073
C01371=1015.976,328.584,352.986,170.418,51.465,160.072
C01372=1015.969,328.337,353.019,170.411,51.469,160.072
C01373=1015.963,328.089,353.054,170.405,51.474,160.072
C01374=1015.956,327.841,353.089,170.398,51.478,160.072
C01375=1015.949,327.594,353.123,170.391,51.482,160.071
C01376=1015.943,327.346,353.157,170.384,51.486,160.071
C01377=1015.937,327.098,353.191,170.377,51.490,160.071
C01378=1015.929,326.851,353.226,170.370,51.495,160.071
C01379=1015.923,326.603,353.260,170.364,51.499,160.070
C01380=1015.917,326.356,353.294,170.356,51.504,160.070
C01381=1015.910,326.108,353.328,170.350,51.507,160.070
C01382=1015.903,325.860,353.362,170.343,51.512,160.070
C01383=1015.897,325.614,353.396,170.336,51.517,160.070
C01384=1015.889,325.366,353.430,170.329,51.521,160.069
C01385=1015.882,325.118,353.463,170.323,51.525,160.069
C01386=1015.876,324.871,353.497,170.316,51.530,160.069
C01387=1015.869,324.623,353.531,170.309,51.534,160.069
C01388=1015.862,324.375,353.564,170.302,51.539,160.068
C01389=1015.856,324.128,353.598,170.295,51.544,160.068
C01390=1015.848,323.880,353.632,170.289,51.547,160.068
C01391=1015.842,323.632,353.666,170.282,51.552,160.068
C01392=1015.836,323.385,353.699,170.276,51.557,160.068
C01393=1015.829,323.107,353.737,170.267,51.562,160.067
C01394=1015.821,322.829,353.774,170.261,51.567,160.067
C01395=1015.813,322.551,353.812,170.253,51.572,160.067
C01396=1015.805,322.273,353.850,170.245,51.577,160.067
C01397=1015.799,322.025,353.883,170.238,51.582,160.067
C01398=1015.792,321.778,353.917,170.233,51.587,160.067
C01399=1015.786,321.531,353.950,170.225,51.591,160.067
C01400=1015.779,321.282,353.984,170.219,51.596,160.066
C01401=1015.772,321.035,354.017,170.212,51.601,160.066
C01402=1015.766,320.787,354.051,170.206,51.605,160.066
C01403=1015.759,320.540,354.084,170.199,51.609,160.066
C01404=1015.753,320.292,354.117,170.192,51.614,160.066
C01405=1015.746,320.044,354.151,170.185,51.619,160.066
C01406=1015.740,319.797,354.184,170.180,51.624,160.066
C01407=1015.733,319.549,354.218,170.173,51.629,160.066
C01408=1015.727,319.301,354.251,170.166,51.633,160.065
C01409=1015.720,319.054,354.284,170.159,51.638,160.065
C01410=1015.713,318.806,354.317,170.153,51.642,160.065
C01411=1015.708,318.558,354.351,170.146,51.647,160.065
C01412=1015.700,318.310,354.384,170.140,51.652,160.065
C01413=1015.694,318.063,354.417,170.133,51.657,160.065
C01414=1015.688,317.815,354.450,170.127,51.661,160.065
C01415=1015.681,317.568,354.483,170.120,51.666,160.065
C01416=1015.675,317.320,354.517,170.114,51.671,160.065
C01417=1015.669,317.072,354.550,170.108,51.676,160.065
C01418=1015.663,316.824,354.583,170.101,51.681,160.065
C01419=1015.655,316.577,354.616,170.094,51.686,160.064
C01420=1015.649,316.329,354.649,170.087,51.691,160.064
C01421=1015.644,316.081,354.682,170.082,51.695,160.064
C01422=1015.637,315.834,354.715,170.075,51.700,160.064
C01423=1015.631,315.586,354.748,170.068,51.705,160.064
C01424=1015.624,315.338,354.782,170.062,51.709,160.064
C01425=1015.617,315.091,354.814,170.056,51.714,160.064
C01426=1015.612,314.843,354.848,170.049,51.719,160.064
C01427=1015.606,314.595,354.881,170.042,51.724,160.064
C01428=1015.599,314.348,354.913,170.037,51.729,160.064
C01429=1015.593,314.100,354.946,170.030,51.734,160.064
C01430=1015.586,313.852,354.979,170.023,51.739,160.064
C01431=1015.581,313.604,355.012,170.017,51.744,160.064
C01432=1015.574,313.356,355.045,170.011,51.749,160.063
C01433=1015.568,313.109,355.078,170.004,51.754,160.064
C01434=1015.562,312.861,355.111,169.999,51.759,160.064
C01435=1015.555,312.614,355.143,169.992,51.764,160.063
C01436=1015.550,312.366,355.177,169.985,51.769,160.063
C01437=1015.544,312.118,355.210,169.980,51.774,160.064
C01438=1015.537,311.871,355.242,169.973,51.779,160.063
C01439=1015.531,311.623,355.275,169.966,51.784,160.063
C01440=1015.525,311.375,355.308,169.961,51.789,160.064
C01441=1015.519,311.127,355.340,169.954,51.794,160.063
C01442=1015.513,310.879,355.373,169.947,51.799,160.063
C01443=1015.507,310.632,355.406,169.942,51.804,160.063
C01444=1015.501,310.384,355.439,169.935,51.809,160.063
C01445=1015.494,310.136,355.471,169.929,51.814,160.063
C01446=1015.488,309.888,355.503,169.923,51.819,160.063
C01447=1015.483,309.640,355.537,169.917,51.824,160.064
C01448=1015.476,309.393,355.569,169.910,51.829,160.063
C01449=1015.470,309.146,355.601,169.904,51.835,160.063
C01450=1015.464,308.898,355.633,169.898,51.840,160.063
C01451=1015.457,308.650,355.665,169.892,51.845,160.064
C01452=1015.451,308.402,355.697,169.885,51.851,160.064
C01453=1015.444,308.130,355.732,169.878,51.857,160.064
C01454=1015.436,307.858,355.768,169.872,51.862,160.064
C01455=1015.430,307.585,355.803,169.864,51.868,160.064
C01456=1015.423,307.312,355.838,169.858,51.874,160.064
C01457=1015.417,307.064,355.870,169.852,51.879,160.064
C01458=1015.410,306.817,355.902,169.845,51.885,160.064
C01459=1015.404,306.569,355.934,169.839,51.891,160.064
C01460=1015.397,306.321,355.965,169.834,51.896,160.064
C01461=1015.391,306.073,355.997,169.827,51.901,160.064
C01462=1015.385,305.825,356.029,169.821,51.907,160.065
C01463=1015.379,305.578,356.061,169.814,51.912,160.064
C01464=1015.372,305.330,356.093,169.808,51.918,160.064
C01465=1015.366,305.082,356.125,169.803,51.923,160.065
C01466=1015.359,304.834,356.156,169.796,51.928,160.065
C01467=1015.353,304.586,356.188,169.790,51.934,160.065
C01468=1015.347,304.338,356.219,169.784,51.940,160.065
C01469=1015.341,304.090,356.251,169.777,51.945,160.065
C01470=1015.335,303.842,356.283,169.772,51.950,160.065
C01471=1015.329,303.594,356.315,169.766,51.956,160.065
C01472=1015.323,303.347,356.347,169.759,51.962,160.065
C01473=1015.316,303.099,356.379,169.753,51.967,160.066
C01474=1015.311,302.850,356.410,169.748,51.972,160.066
C01475=1015.304,302.603,356.441,169.742,51.979,160.066
C01476=1015.298,302.355,356.473,169.735,51.984,160.066
C01477=1015.292,302.107,356.504,169.729,51.990,160.066
C01478=1015.286,301.859,356.536,169.723,51.996,160.066
C01479=1015.280,301.612,356.567,169.717,52.001,160.066
C01480=1015.274,301.363,356.599,169.711,52.006,160.067
C01481=1015.267,301.116,356.631,169.705,52.012,160.067
C01482=1015.262,300.868,356.663,169.699,52.018,160.067
C01483=1015.256,300.620,356.695,169.693,52.024,160.067
C01484=1015.249,300.373,356.726,169.687,52.029,160.067
C01485=1015.244,300.124,356.757,169.681,52.035,160.067
C01486=1015.237,299.876,356.788,169.674,52.040,160.067
C01487=1015.232,299.628,356.820,169.670,52.046,160.068
C01488=1015.225,299.380,356.851,169.663,52.052,160.068
C01489=1015.220,299.132,356.882,169.657,52.058,160.068
C01490=1015.213,298.884,356.914,169.651,52.064,160.068
C01491=1015.208,298.637,356.946,169.645,52.069,160.068
C01492=1015.201,298.389,356.977,169.639,52.075,160.069
C01493=1015.196,298.141,357.008,169.633,52.081,160.069
C01494=1015.189,297.893,357.039,169.627,52.087,160.069
C01495=1015.184,297.646,357.071,169.621,52.092,160.069
C01496=1015.177,297.397,357.102,169.616,52.098,160.069
C01497=1015.172,297.149,357.133,169.610,52.104,160.070
C01498=1015.166,296.901,357.164,169.604,52.110,160.070
C01499=1015.160,296.653,357.196,169.597,52.116,160.070
C01500=1015.154,296.405,357.228,169.592,52.121,160.070
C01501=1015.148,296.157,357.258,169.586,52.127,160.070
C01502=1015.142,295.909,357.290,169.580,52.133,160.071
C01503=1015.137,295.661,357.321,169.574,52.139,160.071
C01504=1015.131,295.414,357.352,169.568,52.145,160.071
C01505=1015.125,295.165,357.383,169.563,52.151,160.071
C01506=1015.119,294.918,357.415,169.556,52.156,160.071
C01507=1015.113,294.669,357.445,169.551,52.163,160.072
C01508=1015.108,294.422,357.477,169.545,52.169,160.072
C01509=1015.102,294.174,357.507,169.539,52.174,160.072
C01510=1015.096,293.926,357.539,169.534,52.181,160.072
C01511=1015.090,293.678,357.570,169.527,52.186,160.073
C01512=1015.085,293.430,357.601,169.521,52.192,160.073
C01513=1015.079,293.175,357.633,169.515,52.199,160.073
C01514=1015.073,292.921,357.665,169.509,52.204,160.073
C01515=1015.067,292.666,357.696,169.504,52.210,160.074
C01516=1015.060,292.412,357.728,169.497,52.217,160.074
C01517=1015.054,292.164,357.758,169.492,52.223,160.074
C01518=1015.049,291.916,357.789,169.487,52.229,160.075
C01519=1015.043,291.667,357.820,169.481,52.236,160.075
C01520=1015.037,291.420,357.850,169.475,52.242,160.075
C01521=1015.031,291.172,357.881,169.468,52.248,160.075
C01522=1015.025,290.924,357.911,169.463,52.254,160.076
C01523=1015.020,290.675,357.942,169.458,52.260,160.076
C01524=1015.014,290.427,357.973,169.452,52.266,160.076
C01525=1015.008,290.179,358.003,169.446,52.272,160.077
C01526=1015.002,289.932,358.033,169.440,52.279,160.077
C01527=1014.996,289.683,358.064,169.434,52.285,160.077
C01528=1014.990,289.435,358.095,169.428,52.291,160.077
C01529=1014.984,289.187,358.125,169.422,52.298,160.078
C01530=1014.978,288.940,358.155,169.417,52.304,160.078
C01531=1014.972,288.691,358.186,169.412,52.310,160.078
C01532=1014.966,288.443,358.216,169.406,52.316,160.079
C01533=1014.961,288.195,358.246,169.400,52.323,160.079
C01534=1014.955,287.947,358.276,169.394,52.329,160.079
C01535=1014.949,287.699,358.307,169.389,52.336,160.080
C01536=1014.943,287.451,358.337,169.383,52.342,160.080
C01537=1014.937,287.203,358.368,169.377,52.349,160.080
C01538=1014.931,286.954,358.397,169.371,52.355,160.081
C01539=1014.926,286.707,358.428,169.366,52.361,160.081
C01540=1014.920,286.459,358.458,169.360,52.367,160.081
C01541=1014.914,286.211,358.488,169.355,52.374,160.082
C01542=1014.908,285.962,358.518,169.349,52.381,160.082
C01543=1014.903,285.715,358.548,169.343,52.387,160.083
C01544=1014.897,285.466,358.578,169.337,52.393,160.083
C01545=1014.891,285.218,358.608,169.332,52.400,160.083
C01546=1014.885,284.971,358.639,169.326,52.407,160.084
C01547=1014.880,284.722,358.668,169.320,52.413,160.084
C01548=1014.873,284.474,358.699,169.315,52.420,160.084
C01549=1014.867,284.225,358.728,169.310,52.426,160.085
C01550=1014.861,283.978,358.758,169.304,52.432,160.085
C01551=1014.856,283.729,358.788,169.299,52.439,160.086
C01552=1014.850,283.481,358.818,169.293,52.446,160.086
C01553=1014.844,283.233,358.847,169.287,52.453,160.086
C01554=1014.838,282.985,358.878,169.281,52.459,160.087
C01555=1014.833,282.737,358.907,169.276,52.466,160.087
C01556=1014.827,282.489,358.937,169.270,52.473,160.088
C01557=1014.820,282.241,358.967,169.265,52.480,160.088
C01558=1014.815,281.993,358.996,169.259,52.486,160.088
C01559=1014.809,281.744,359.026,169.253,52.493,160.089
C01560=1014.803,281.497,359.056,169.248,52.499,160.089
C01561=1014.798,281.249,359.085,169.242,52.506,160.090
C01562=1014.792,281.000,359.115,169.237,52.513,160.090
C01563=1014.787,280.752,359.144,169.231,52.520,160.090
C01564=1014.780,280.505,359.174,169.225,52.527,160.091
C01565=1014.775,280.256,359.204,169.220,52.533,160.091
C01566=1014.769,280.008,359.233,169.214,52.540,160.092
C01567=1014.763,279.760,359.262,169.209,52.547,160.092
C01568=1014.758,279.511,359.292,169.203,52.554,160.093
C01569=1014.753,279.266,359.322,169.198,52.561,160.093
C01570=1014.746,279.021,359.351,169.192,52.568,160.094
C01571=1014.740,278.776,359.380,169.187,52.574,160.094
C01572=1014.736,278.530,359.409,169.182,52.581,160.095
C01573=1014.729,278.285,359.438,169.176,52.588,160.095
C01574=1014.724,278.040,359.468,169.171,52.594,160.095
C01575=1014.718,277.795,359.497,169.165,52.601,160.096
C01576=1014.713,277.550,359.525,169.160,52.608,160.096
C01577=1014.708,277.302,359.555,169.154,52.615,160.097
C01578=1014.701,277.053,359.584,169.149,52.622,160.097
C01579=1014.696,276.806,359.613,169.143,52.629,160.098
C01580=1014.691,276.557,359.643,169.138,52.636,160.098
C01581=1014.685,276.309,359.673,169.132,52.643,160.099
C01582=1014.679,276.061,359.702,169.127,52.650,160.099
C01583=1014.674,275.813,359.731,169.122,52.657,160.100
C01584=1014.668,275.565,359.760,169.116,52.664,160.100
C01585=1014.662,275.316,359.790,169.111,52.671,160.101
C01586=1014.656,275.068,359.819,169.105,52.678,160.101
C01587=1014.651,274.820,359.848,169.100,52.685,160.102
C01588=1014.645,274.572,359.876,169.095,52.692,160.102
C01589=1014.640,274.323,359.906,169.089,52.699,160.103
C01590=1014.634,274.075,359.935,169.084,52.706,160.103
C01591=1014.628,273.828,359.964,169.078,52.713,160.104
C01592=1014.623,273.579,359.992,169.073,52.721,160.104
C01593=1014.616,273.331,360.021,169.068,52.728,160.105
C01594=1014.612,273.083,360.051,169.062,52.735,160.105
C01595=1014.606,272.834,360.079,169.057,52.742,160.106
C01596=1014.600,272.586,360.109,169.050,52.749,160.106
C01597=1014.594,272.338,360.137,169.045,52.756,160.107
C01598=1014.589,272.089,360.166,169.040,52.764,160.107
C01599=1014.583,271.841,360.195,169.035,52.771,160.108
C01600=1014.578,271.593,360.223,169.029,52.778,160.108
C01601=1014.572,271.344,360.253,169.024,52.785,160.109
C01602=1014.566,271.096,360.282,169.019,52.792,160.109
C01603=1014.561,270.848,360.311,169.014,52.800,160.110
C01604=1014.555,270.600,360.340,169.008,52.807,160.111
C01605=1014.550,270.352,360.368,169.003,52.814,160.111
C01606=1014.544,270.103,360.397,168.998,52.822,160.112
C01607=1014.539,269.855,360.425,168.992,52.830,160.112
C01608=1014.533,269.607,360.454,168.986,52.837,160.113
C01609=1014.527,269.358,360.483,168.981,52.844,160.114
C01610=1014.522,269.110,360.511,168.976,52.852,160.114
C01611=1014.516,268.862,360.540,168.970,52.859,160.115
C01612=1014.511,268.614,360.569,168.966,52.866,160.115
C01613=1014.505,268.365,360.598,168.960,52.874,160.116
C01614=1014.500,268.117,360.626,168.955,52.881,160.117
C01615=1014.494,267.869,360.654,168.949,52.889,160.117
C01616=1014.489,267.620,360.683,168.944,52.897,160.118
C01617=1014.483,267.372,360.712,168.939,52.904,160.118
C01618=1014.477,267.124,360.740,168.934,52.911,160.119
C01619=1014.472,266.875,360.768,168.928,52.919,160.119
C01620=1014.466,266.627,360.796,168.923,52.926,160.120
C01621=1014.461,266.379,360.825,168.917,52.934,160.121
C01622=1014.455,266.131,360.853,168.912,52.942,160.121
C01623=1014.449,265.882,360.882,168.907,52.949,160.122
C01624=1014.444,265.634,360.910,168.902,52.957,160.123
C01625=1014.438,265.385,360.938,168.897,52.964,160.123
C01626=1014.434,265.137,360.967,168.892,52.971,160.124
C01627=1014.428,264.889,360.995,168.886,52.980,160.124
C01628=1014.422,264.641,361.024,168.880,52.987,160.125
C01629=1014.417,264.397,361.050,168.875,52.995,160.126
C01630=1014.412,264.155,361.078,168.870,53.002,160.126
C01631=1014.406,263.911,361.106,168.865,53.009,160.127
C01632=1014.400,263.669,361.133,168.860,53.017,160.128
C01633=1014.395,263.426,361.160,168.855,53.024,160.128
C01634=1014.390,263.183,361.188,168.850,53.032,160.129
C01635=1014.384,262.941,361.215,168.845,53.040,160.130
C01636=1014.378,262.697,361.243,168.840,53.047,160.130
C01637=1014.373,262.449,361.271,168.834,53.055,160.131
C01638=1014.368,262.201,361.299,168.829,53.063,160.131
C01639=1014.362,261.952,361.327,168.824,53.071,160.132
C01640=1014.357,261.704,361.355,168.819,53.079,160.133
C01641=1014.351,261.456,361.383,168.813,53.087,160.133
C01642=1014.345,261.207,361.411,168.808,53.094,160.134
C01643=1014.340,260.959,361.439,168.803,53.102,160.135
C01644=1014.335,260.711,361.467,168.798,53.110,160.135
C01645=1014.329,260.462,361.495,168.792,53.118,160.136
C01646=1014.324,260.213,361.522,168.787,53.126,160.137
C01647=1014.318,259.965,361.550,168.782,53.134,160.137
C01648=1014.313,259.717,361.578,168.778,53.141,160.138
C01649=1014.308,259.468,361.607,168.772,53.150,160.139
C01650=1014.302,259.220,361.634,168.767,53.157,160.140
C01651=1014.297,258.972,361.662,168.762,53.165,160.140
C01652=1014.291,258.724,361.689,168.756,53.174,160.141
C01653=1014.286,258.475,361.716,168.752,53.182,160.142
C01654=1014.279,258.227,361.744,168.747,53.190,160.143
C01655=1014.274,257.978,361.771,168.741,53.198,160.143
C01656=1014.268,257.730,361.799,168.736,53.206,160.144
C01657=1014.263,257.482,361.826,168.730,53.214,160.145
C01658=1014.257,257.232,361.854,168.726,53.223,160.146
C01659=1014.251,256.985,361.881,168.721,53.231,160.146
C01660=1014.246,256.736,361.908,168.715,53.239,160.147
C01661=1014.241,256.488,361.936,168.710,53.247,160.148
C01662=1014.235,256.240,361.963,168.705,53.256,160.148
C01663=1014.229,255.990,361.990,168.700,53.263,160.149
C01664=1014.224,255.742,362.018,168.694,53.272,160.150
C01665=1014.218,255.494,362.045,168.689,53.280,160.151
C01666=1014.213,255.246,362.073,168.685,53.288,160.151
C01667=1014.207,254.997,362.100,168.679,53.296,160.152
C01668=1014.202,254.749,362.127,168.674,53.305,160.153
C01669=1014.196,254.499,362.155,168.668,53.313,160.154
C01670=1014.190,254.252,362.182,168.664,53.321,160.154
C01671=1014.185,254.003,362.209,168.658,53.330,160.155
C01672=1014.179,253.755,362.236,168.653,53.338,160.156
C01673=1014.174,253.507,362.264,168.649,53.346,160.157
C01674=1014.168,253.258,362.290,168.643,53.354,160.158
C01675=1014.163,253.010,362.318,168.639,53.363,160.158
C01676=1014.158,252.761,362.345,168.633,53.371,160.159
C01677=1014.152,252.513,362.372,168.628,53.380,160.160
C01678=1014.147,252.264,362.399,168.623,53.388,160.161
C01679=1014.141,252.016,362.426,168.618,53.396,160.161
C01680=1014.136,251.767,362.453,168.612,53.405,160.162
C01681=1014.131,251.518,362.481,168.608,53.413,160.163
C01682=1014.125,251.270,362.508,168.602,53.422,160.164
C01683=1014.120,251.021,362.535,168.598,53.430,160.165
C01684=1014.114,250.773,362.562,168.593,53.438,160.165
C01685=1014.109,250.525,362.589,168.587,53.447,160.166
C01686=1014.104,250.276,362.617,168.583,53.455,160.167
C01687=1014.098,250.028,362.643,168.577,53.464,160.168
C01688=1014.093,249.779,362.671,168.573,53.473,160.169
C01689=1014.088,249.535,362.697,168.567,53.481,160.169
C01690=1014.083,249.292,362.723,168.562,53.489,160.170
C01691=1014.078,249.047,362.750,168.558,53.497,160.171
C01692=1014.072,248.804,362.776,168.552,53.506,160.172
C01693=1014.066,248.560,362.803,168.548,53.514,160.173
C01694=1014.062,248.316,362.829,168.543,53.523,160.174
C01695=1014.057,248.072,362.855,168.537,53.531,160.174
C01696=1014.051,247.828,362.882,168.533,53.540,160.175
C01697=1014.046,247.579,362.909,168.527,53.548,160.176
C01698=1014.040,247.331,362.936,168.523,53.557,160.177
C01699=1014.036,247.083,362.963,168.517,53.565,160.178
C01700=1014.030,246.835,362.990,168.513,53.574,160.179
C01701=1014.025,246.586,363.017,168.507,53.582,160.179
C01702=1014.020,246.337,363.044,168.503,53.591,160.180
C01703=1014.015,246.088,363.070,168.498,53.600,160.181
C01704=1014.010,245.840,363.097,168.493,53.609,160.182
C01705=1014.004,245.591,363.124,168.487,53.617,160.183
C01706=1013.999,245.343,363.151,168.483,53.625,160.184
C01707=1013.994,245.095,363.178,168.478,53.634,160.184
C01708=1013.989,244.846,363.205,168.473,53.643,160.185
C01709=1013.984,244.597,363.231,168.468,53.652,160.186
C01710=1013.978,244.349,363.258,168.464,53.661,160.187
C01711=1013.974,244.101,363.285,168.458,53.670,160.188
C01712=1013.968,243.852,363.311,168.454,53.678,160.189
C01713=1013.963,243.604,363.339,168.448,53.687,160.190
C01714=1013.958,243.354,363.365,168.444,53.695,160.190
C01715=1013.952,243.106,363.392,168.439,53.704,160.191
C01716=1013.948,242.858,363.419,168.433,53.713,160.192
C01717=1013.942,242.610,363.445,168.429,53.722,160.193
C01718=1013.937,242.360,363.472,168.423,53.731,160.194
C01719=1013.932,242.113,363.498,168.419,53.739,160.195
C01720=1013.927,241.864,363.524,168.414,53.749,160.196
C01721=1013.921,241.615,363.551,168.409,53.758,160.197
C01722=1013.917,241.367,363.577,168.405,53.767,160.198
C01723=1013.911,241.119,363.603,168.399,53.776,160.199
C01724=1013.906,240.870,363.629,168.394,53.785,160.199
C01725=1013.901,240.621,363.657,168.390,53.794,160.200
C01726=1013.896,240.373,363.682,168.384,53.803,160.201
C01727=1013.890,240.124,363.709,168.379,53.812,160.202
C01728=1013.885,239.875,363.735,168.375,53.820,160.203
C01729=1013.880,239.627,363.762,168.370,53.830,160.204
C01730=1013.875,239.378,363.788,168.365,53.839,160.205
C01731=1013.869,239.130,363.814,168.360,53.848,160.206
C01732=1013.865,238.881,363.840,168.355,53.857,160.207
C01733=1013.859,238.632,363.866,168.350,53.866,160.208
C01734=1013.853,238.384,363.893,168.345,53.875,160.209
C01735=1013.849,238.136,363.919,168.341,53.884,160.210
C01736=1013.843,237.887,363.944,168.336,53.894,160.211
C01737=1013.838,237.639,363.971,168.330,53.903,160.212
C01738=1013.832,237.390,363.997,168.325,53.912,160.212
C01739=1013.827,237.141,364.023,168.321,53.921,160.214
C01740=1013.822,236.893,364.048,168.316,53.930,160.214
C01741=1013.817,236.644,364.074,168.311,53.940,160.216
C01742=1013.811,236.395,364.100,168.306,53.949,160.216
C01743=1013.806,236.147,364.126,168.301,53.959,160.217
C01744=1013.801,235.898,364.152,168.297,53.968,160.218
C01745=1013.796,235.650,364.178,168.292,53.977,160.220
C01746=1013.790,235.401,364.204,168.287,53.986,160.220
C01747=1013.785,235.153,364.229,168.282,53.996,160.221
C01748=1013.780,234.904,364.255,168.277,54.005,160.222
C01749=1013.775,234.657,364.281,168.272,54.015,160.223
C01750=1013.769,234.409,364.307,168.267,54.024,160.224
C01751=1013.764,234.162,364.332,168.263,54.033,160.225
C01752=1013.759,233.915,364.358,168.257,54.042,160.226
C01753=1013.753,233.667,364.383,168.253,54.052,160.227
C01754=1013.749,233.420,364.409,168.247,54.061,160.228
C01755=1013.743,233.172,364.434,168.243,54.071,160.229
C01756=1013.739,232.925,364.460,168.239,54.080,160.230
C01757=1013.733,232.676,364.486,168.233,54.090,160.231
C01758=1013.728,232.428,364.512,168.229,54.099,160.232
C01759=1013.723,232.179,364.538,168.224,54.109,160.233
C01760=1013.718,231.930,364.563,168.219,54.118,160.234
C01761=1013.713,231.681,364.588,168.214,54.128,160.235
C01762=1013.707,231.433,364.613,168.210,54.137,160.237
C01763=1013.702,231.185,364.639,168.205,54.146,160.237
C01764=1013.697,230.936,364.665,168.200,54.156,160.238
C01765=1013.692,230.688,364.691,168.195,54.166,160.240
C01766=1013.686,230.439,364.716,168.190,54.176,160.241
C01767=1013.682,230.191,364.742,168.185,54.185,160.241
C01768=1013.676,229.941,364.767,168.180,54.195,160.243
C01769=1013.672,229.693,364.793,168.176,54.205,160.244
C01770=1013.667,229.444,364.818,168.171,54.214,160.245
C01771=1013.661,229.195,364.844,168.166,54.223,160.246
C01772=1013.656,228.947,364.869,168.161,54.233,160.247
C01773=1013.651,228.699,364.894,168.156,54.243,160.248
C01774=1013.646,228.450,364.920,168.151,54.253,160.249
C01775=1013.641,228.201,364.945,168.147,54.263,160.250
C01776=1013.636,227.952,364.971,168.142,54.272,160.251
C01777=1013.630,227.704,364.996,168.137,54.282,160.252
C01778=1013.625,227.455,365.021,168.132,54.292,160.253
C01779=1013.620,227.206,365.047,168.128,54.302,160.254
C01780=1013.615,226.958,365.072,168.123,54.312,160.255
C01781=1013.611,226.709,365.097,168.118,54.322,160.256
C01782=1013.604,226.460,365.122,168.113,54.331,160.257
C01783=1013.600,226.211,365.147,168.109,54.341,160.258
C01784=1013.595,225.963,365.173,168.104,54.351,160.260
C01785=1013.590,225.714,365.197,168.099,54.361,160.261
C01786=1013.584,225.465,365.223,168.094,54.371,160.262
C01787=1013.579,225.217,365.247,168.090,54.381,160.263
C01788=1013.574,224.968,365.273,168.085,54.390,160.264
C01789=1013.565,224.568,365.313,168.077,54.407,160.266
C01790=1013.557,224.167,365.352,168.070,54.423,160.268
C01791=1013.549,223.766,365.393,168.062,54.439,160.269
C01792=1013.541,223.365,365.433,168.054,54.455,160.271
C01793=1013.535,223.116,365.457,168.050,54.466,160.272
C01794=1013.530,222.868,365.483,168.045,54.475,160.273
C01795=1013.524,222.619,365.508,168.040,54.485,160.274
C01796=1013.520,222.370,365.533,168.036,54.495,160.276
C01797=1013.515,222.122,365.558,168.031,54.506,160.277
C01798=1013.510,221.873,365.582,168.026,54.516,160.278
C01799=1013.505,221.624,365.607,168.021,54.526,160.279
C01800=1013.499,221.375,365.632,168.017,54.536,160.280
C01801=1013.494,221.127,365.657,168.012,54.546,160.281
C01802=1013.489,220.878,365.682,168.007,54.556,160.282
C01803=1013.485,220.629,365.706,168.003,54.566,160.283
C01804=1013.479,220.381,365.731,167.997,54.577,160.285
C01805=1013.475,220.132,365.756,167.993,54.587,160.286
C01806=1013.469,219.883,365.781,167.989,54.597,160.287
C01807=1013.464,219.634,365.806,167.984,54.607,160.288
C01808=1013.459,219.386,365.830,167.979,54.617,160.289
C01809=1013.452,219.034,365.865,167.973,54.632,160.291
